VAR_INST
	r_Soc							: REAL;
	fb_SOCLowLimit					: fbValueOutOfRange;
	fb_SOCHighLimit					: fbValueOutOfRange;
	r_SoCMinActual 					: REAL;
	r_SoCMaxActual					: REAL;
	r_deltaSoC						: REAL;
	r_ratio							: REAL;
	r_offset						: REAL;
	
	RS_chargingAllowed				: RS;
	RS_DischargingAllowed			: RS;
END_VAR
//Calculations
r_deltaSoC:= st_params.r_SoCAbsoluteMax - st_params.r_SoCAbsoluteMin;
r_ratio := 1 / SEL(r_deltaSoC=0,r_deltaSoC/100,1);
r_offset := st_params.r_SoCAbsoluteMin * r_Ratio;


//user soc setpoint, first limit user value with 100% and scale to original battery soc 
r_SoCMinActual := (LIMIT(0, set.r_SocMin, set.r_SocMax) + r_Offset) / r_ratio;
r_SoCMaxActual := sel(AutoSOCCalibrationRequired,(LIMIT(set.r_SocMin,set.r_SocMax,100) + r_Offset) / r_ratio, 100);

//Set limit with error when hard limits exceed absolute VDL limits
fb_SOCLowLimit(
	r_var		:= r_SocMinActual, 
	r_min		:= st_params.r_SoCAbsoluteMin, 
	r_max		:= st_params.r_SoCAbsoluteMax,
	r_WhenError := st_params.r_SoCAbsoluteMin,
	b_IsError	=> get.events.b_SoCLowLimitOutOfRange);

fb_SOCHighLimit(
	r_var		:= r_SocMaxActual, 
	r_min		:= st_params.r_SoCAbsoluteMin, 
	r_max		:= st_params.r_SoCAbsoluteMax,
	r_WhenError := st_params.r_SoCAbsoluteMin,
	b_IsError	=> get.events.b_SoCHighLimitOutOfRange);


//Set scaled soc to monitoring
get.BatteryInfo.r_SOCScaled := F_RoundReal(LIMIT(0, get.BatteryInfo.r_SOC * r_ratio - r_offset, 100),1); // set limit to avoid exceed 0 or 100%.

//set scaled kwh discharging remaining
get.BatteryInfo.r_RemainingDischargeEnergyNett := r_deltaSoC/ 100 * get.BatteryInfo.r_RemainingDischargeEnergy;
get.BatteryInfo.r_RemainingChargeEnergyNett := r_deltaSoC/ 100 * get.BatteryInfo.r_RemainingChargeEnergy;

r_Soc := get.BatteryInfo.r_SoC;
//Set Charge only when soft high limit reached
rs_dischargingAllowed(
	set:=r_SoC > (r_SoCMinActual + st_params.r_SocHysteresis),
	Reset1 := r_SoC <= r_SoCMinActual OR get.BatteryInfo.e_BMS_Status = eBMS_Status.FullDischarge,
	Q1 => get.BatteryInfo.b_dischargingAllowed);

//Set discharge only when soft high limit reached
rs_chargingAllowed(
	SET:= r_SoC < (r_SoCMaxActual - st_params.r_SocHysteresis),
	RESET1:= r_SoC >= r_SoCMaxActual OR get.BatteryInfo.e_BMS_Status = eBMS_Status.FullCharge,
	Q1=> get.BatteryInfo.b_chargingAllowed);
END_METHOD

METHOD PRIVATE CalculateTimeRemaining : BOOL
VAR_INPUT
END_VAR

VAR_OUTPUT
END_VAR

VAR_INST
	a_PowerArray			: ARRAY [1..20] OF REAL;
	st_Params_MA			: ST_CTRL_MOVING_AVERAGE_PARAMS;
	ui_filterSize			: UINT := 10;
	fb_SmoothPower			: FB_CTRL_MOVING_AVERAGE;
	r_PowerMA				: REAL;
	r_HoursRemaining		: REAL;
END_VAR
//SMOOTH SETPOINT VALUE SINCE VALUE IS SWITCHED RAPIDLY BETWEEN UPPER AND LOWER GRID LIMIT.
st_Params_MA.tCtrlCycleTime := T#100MS;
	st_Params_MA.tTaskCycleTime := T#1MS;
	st_Params_MA.nWorkArray_SIZEOF := SIZEOF(a_PowerArray);
	st_Params_MA.pWorkArray_ADR	:= ADR(a_PowerArray);
	st_Params_MA.nSamplesToFilter:= ui_filterSize;

fb_SmoothPower(fin:= get.BatteryInfo.r_SystemPower,
				eMode := E_CTRL_MODE.eCTRL_MODE_ACTIVE,
				fout=> r_PowerMA,
				stParams := st_Params_MA);
				
r_HoursRemaining := get.BatteryInfo.r_RemainingDischargeEnergyNett / MAX(1, r_PowerMA);
END_METHOD

METHOD PRIVATE ClearBMSFaults : BOOL
VAR_IN_OUT CONSTANT
	st_params			: ST_BMS_params;
END_VAR

VAR_INST
	WriteRegSet		:	FB_MBWriteSingleReg;
	WriteRegClear	:	FB_MBWriteSingleReg;
	
	bCommBusy	:	BOOL;
	bComError	:	BOOL;
	errID		:	UDINT;
	b_ClearDone	:	BOOL := FALSE;

	w_ClearFault	:	WORD;
	TX1Done 	: 	f_trig;
	
	bCommBusy2	:	BOOL;
	bComError2	:	BOOL;
	errID2		:	UDINT;
	TX2Done 	: 	f_trig;

	ComRetryCounter	:	USINT := 0;	
	
	ResetDelayTimer	: Tp := (PT:=T#500MS);
END_VAR
//Catl says we need to write 1 to clear, then write back to 0 to be able to log new errors.
//This method is called continuously when bms is active. It will usually write zero's.
//If set.b_ClearFault is 1, that will be written. The value will be cleared by this method after the write so next write will be a 0 again.
//With this, a reset cycle takes half a second with the current ComTimer.

ClearBMSFaults := FALSE;

ComTimer(in := NOT(ComTimer.Q OR bCommBusy));

//first write clearing register to 1
WriteRegSet(
	sIPAddr := st_params.IP_BMS,
	nTCPPort := 502,
	nUnitID := 255,//16#FF;
	nMBAddr := 908,
	nValue := 1,
	tTimeOut := t_TimeOut,
	bExecute := ComTimer.Q,
	bBusy => bCommBusy,
	bError => bComError,
	nErrId => errID,
);

TX1Done(CLK := bCommBusy);
b_ClearDone	:= 	TX1Done.Q AND NOT bComError;
ResetDelayTimer(in:=b_ClearDone);
//reset value back to 0 afterwards. CATL requirement
WriteRegClear(
	sIPAddr := st_params.IP_BMS,
	nTCPPort := 502,
	nUnitID := 255,//16#FF;
	nMBAddr := 908,
	nValue := 0,
	tTimeout := T#100MS,
	bExecute := NOT ResetDelayTimer.Q,
	bBusy => bCommBusy2,
	bError => bComError2,
	nErrId => errID2
);

TX2Done(CLK := bCommBusy2);

IF (TX1Done.Q AND bComError) OR (TX2Done.Q AND bComError2) THEN
	ComRetryCounter := ComRetryCounter + 1;
	IF COMRetryCounter > 5 THEN
		b_MBComErrorActive := TRUE;
		ClearBMSFaults := TRUE;
	END_IF
END_IF

IF (TX1Done.Q AND NOT bComError) THEN
	arDatalogEMS[4] := 1;	
END_IF

IF TX2Done.Q AND NOT bComError2 THEN
	arDatalogEMS[4] := 0;	
	b_MBComErrorActive := FALSE;
	ComRetryCounter := 0;
	ClearBMSFaults := TRUE;
END_IF
END_METHOD

METHOD EMSTOP : BOOL
EMSTOP := FALSE;

FBState := ePOUState.EMSTOP;

IF get.MBMU.BatteryStatus.e_BMS_PowerOnStatus <> ePowerOnStatus.On THEN
	EMSTOP := TRUE;
END_IF
END_METHOD

METHOD PRIVATE GetBatteryInfo : BOOL

VAR_IN_OUT
	IN : ST_MBMU_BatterySummary;
	OUT: ST_BMS_BatterySummary;
END_VAR


VAR_INST
	ton_syncPulse : TON := (PT := T#100MS);
	t_SyncTimer	: TIME := T#100MS;
	tof_Release : TOF := (PT:= T#2S);
END_VAR
tof_Release(IN:= get.Events.b_COMMUNICATION_ERROR OR get.MBMU.BatteryStatus.r_SOC > 101);

//set batterysummery data if MBMU gives no shit.
IF ton_syncPulse.Q THEN
	IF NOT tof_Release.Q THEN
		//copy inherited data from original location.
 		MEMCPY(ADR(OUT), ADR(IN), SIZEOF(IN));
		//generate additional data
		CalculateSoCUser(get := get, set := set, st_params:=st_params);
		CalculatedRatings(numberOfStrings:= settings.Configuration.by_NoBatteryStrings);
		CalculateCumulativeValues(get := OUT, t_cycleTime := t_syncTimer);
	ELSE
		out.ar_CellTemperature[0] := -273;
		out.ar_CellTemperature[1] := -273;
		out.ar_CellTemperature[2] := -273;
	END_IF
END_IF
 

ton_syncPulse(IN := NOT ton_syncPulse.Q, PT := t_SyncTimer);
END_METHOD

METHOD PRIVATE GetCellData : BOOL
VAR_IN_OUT CONSTANT
	st_params			: ST_BMS_params;
END_VAR

VAR_INPUT
	SBMUID	:	BYTE;	//SBMU 1-#ofstrings
	CSCID	:	BYTE;	//CSC 1-4
END_VAR

VAR_OUTPUT
	CellVoltages		:	ARRAY[1..52] OF REAL;
	Celltemperatures	:	ARRAY[1..16] OF INT;
	BalanceStatus		:	ARRAY[1..4] OF WORD; //bit per cell?
END_VAR

VAR_INST
	MBReadCellVoltages	: 	FB_MBReadRegs;
	MBReadTemperatures	: 	FB_MBReadRegs;
	MBReadCellBalance	: 	FB_MBReadRegs;
	
//	CellVoltageData		: 	ARRAY[1..52] OF WORD;
	TemperatureData		: 	ARRAY[1..16] OF BYTE;
//	CellBalanceData		: 	ARRAY[1..4] OF WORD;
	
	bCommBusy			:	ARRAY[1..3] OF BOOL;
	bComError			:	ARRAY[1..3] OF BOOL;
	errID				:	ARRAY[1..3] OF UDINT;
	cbRead				:	ARRAY[1..3] OF UDINT;
	TransmissionDone	: 	ARRAY[1..3] OF f_trig;
	
	DataComplete		:	ARRAY[1..3] OF BOOL;
	
	//ComTimer			:	Ton := (PT := TIME#0S500MS);
END_VAR

VAR
	LoopCounter			:	INT;
END_VAR

GetCellData := FALSE;

IF (SBMUID < 1) OR (SBMUID > get.MBMU.by_NumberOfSubSystems) THEN
	GetCellData := TRUE;
	RETURN;
END_IF
IF (CSCID < 1) OR (CSCID > 4) THEN
	GetCellData := TRUE;
	RETURN;
END_IF

ComTimer(in := NOT(ComTimer.Q OR bCommBusy[1] OR bCommBusy[2] OR bCommBusy[3]));

IF ComTimer.Q THEN
	DataComplete[1] := FALSE;
	DataComplete[2] := FALSE;
	DataComplete[3] := FALSE;
END_IF

MBReadCellVoltages(
sIPAddr := st_params.IP_BMS,
nTCPPort := 502,
nUnitID := 255,//16#FF;
nMBAddr := (SBMUID*1024)+128+(52*(CSCID-1)),	//SBMU 1, module 1, start at 0x0480, increment 52 per module & 1024 per sbmu
nQuantity := 52,
cbLength := SIZEOF(CellVoltages),
pDestAddr := ADR(CellVoltages),
bExecute := ComTimer.Q,
bBusy => bCommBusy[1],
bError => bComError[1],
nErrId => errID[1],
cbRead => cbRead[1],
tTimeOut := t_TimeOut,
);

MBReadTemperatures(
sIPAddr := st_params.IP_BMS,
nTCPPort := 502,
nUnitID := 1,//16#FF;
nMBAddr := (SBMUID*1024)+704+(8*(CSCID-1)),	//SBMU 1, module 1, start at 0x06c0, increment 8 (16 byte) per module & 1024 per sbmu
nQuantity := 8*2,
cbLength := SIZEOF(TemperatureData),
pDestAddr := ADR(TemperatureData),
bExecute := ComTimer.Q,
bBusy => bCommBusy[2],
bError => bComError[2],
nErrId => errID[2],
cbRead => cbRead[2],
tTimeOut := t_TimeOut,
);

MBReadTemperatures(
sIPAddr := st_params.IP_BMS,
nTCPPort := 502,
nUnitID := 1,//16#FF;
nMBAddr := (SBMUID*1024)+912+(4*(CSCID-1)),	//SBMU 1, module 1, start at 0x0790, increment 4 per module & 1024 per sbmu
											//not sure if CSC2 starts at address 4, or immediatly follows after last cell of csc1.
nQuantity := 4*2,
cbLength := SIZEOF(BalanceStatus),
pDestAddr := ADR(BalanceStatus),
bExecute := ComTimer.Q,
bBusy => bCommBusy[3],
bError => bComError[3],
nErrId => errID[3],
cbRead => cbRead[3],
tTimeOut := t_TimeOut,
);

TransmissionDone[1](clk:=bCommBusy[1]);
TransmissionDone[2](clk:=bCommBusy[2]);
TransmissionDone[3](clk:=bCommBusy[3]);

IF TransmissionDone[1].Q AND NOT bComError[1] THEN
	DataComplete[1] := TRUE;
END_IF

IF TransmissionDone[2].Q AND NOT bComError[2] THEN
	FOR loopcounter := 1 TO 16 BY 1 DO
		Celltemperatures[loopcounter] := TemperatureData[loopcounter]-50;
	END_FOR
	DataComplete[2] := TRUE;
END_IF

IF TransmissionDone[1].Q AND NOT bComError[1] THEN
	DataComplete[3] := TRUE;
END_IF

GetCellData := DataComplete[1] AND DataComplete[2] AND DataComplete[3];
END_METHOD

METHOD GetDiagnostics 
VAR_IN_OUT
	AddError		: ARRAY [*] OF FB_AddErrorST;
	a_ActiveEvents	: ARRAY [*] OF ST_ErrorStruct;
	w_Index			: WORD;
END_VAR
(*BMS errors (sunspec)*)
	(*BMS Communication error*)		AddError[w_Index](
			b_ErrorTrig				:= get.Events.b_COMMUNICATION_ERROR,
			out_ST_Error			:= a_ActiveEvents[w_Index],
			w_ErrorID				:= 1,
			e_ObjectID				:= e_id,						//only first call set object ID.
			s_Message				:= 'communication error',
			e_sev					:= eSeverity.QuickShutdown,	//<-- maybe normal shutdown?
			b_AutoClear				:= FALSE,
			t_TriggerTime			:= TIME#10S,
			e_ErrAckAccess			:= eErrAckAccess.Operator
			);
		w_Index := w_Index +1;
		
	(*Configuration fault*)		AddError[w_Index](
			b_ErrorTrig				:= get.Events.b_CONFIGURATION_ALARM,
			out_ST_Error			:= a_ActiveEvents[w_Index],
			w_ErrorID				:= 2,
			s_Message				:= 'configuration error',
			e_sev					:= eSeverity.NormalShutdown,
			b_AutoClear				:= FALSE,
			e_ErrAckAccess			:= eErrAckAccess.VDL
			//in_t_TriggerTime		:= TIME#500MS,
			//in_e_ErrAckAccess		:= TRUE,
			);
		w_Index := w_Index +1;
	
	(*Configuration warning*)		AddError[w_Index](
			b_ErrorTrig				:= get.Events.b_CONFIGURATION_WARNING,
			out_ST_Error			:= a_ActiveEvents[w_Index],
			w_ErrorID				:= 3,
			s_Message				:= 'configuration error',
			e_sev					:= eSeverity.Warning,
			b_AutoClear				:= FALSE,
			e_ErrAckAccess			:= eErrAckAccess.Operator
			//in_t_TriggerTime		:= TIME#500MS,
			//in_e_ErrAckAccess		:= TRUE,
			);
		w_Index := w_Index +1;
		
	(*Contactor fault*)		AddError[w_Index](
			b_ErrorTrig				:= get.Events.b_CONTACTOR_ERROR,
			out_ST_Error			:= a_ActiveEvents[w_Index],
			w_ErrorID				:= 4,
			s_Message				:= 'contactor fault',
			e_sev					:= eSeverity.QuickShutdown,
			b_AutoClear				:= FALSE,
			e_ErrAckAccess			:= eErrAckAccess.Operator
			//in_t_TriggerTime		:= TIME#500MS,
			//in_e_ErrAckAccess		:= TRUE,
			);
		w_Index := w_Index +1;
		
	(*Current imbalance warning*)		AddError[w_Index](						//unused, will always be false
			b_ErrorTrig				:= get.Events.b_CURRENT_IMBALANCE_WARNING,
			out_ST_Error			:= a_ActiveEvents[w_Index],
			w_ErrorID				:= 5,
			s_Message				:= 'current imbalance warning',
			e_sev					:= eSeverity.Warning,
			b_AutoClear				:= FALSE,
			e_ErrAckAccess			:= eErrAckAccess.General
			//in_t_TriggerTime		:= TIME#500MS,
			);
		w_Index := w_Index +1;
		
	(*Fan error*)		AddError[w_Index](
			b_ErrorTrig				:= get.Events.b_FAN_ERROR,
			out_ST_Error			:= a_ActiveEvents[w_Index],
			w_ErrorID				:= 6,
			s_Message				:= 'fan error',
			e_sev					:= eSeverity.NormalShutdown,
			b_AutoClear				:= FALSE,
			//in_t_TriggerTime		:= TIME#500MS,
			e_ErrAckAccess			:= eErrackAccess.Operator
			);
		w_Index := w_Index +1;

	(*Ground fault*)		AddError[w_Index](
			b_ErrorTrig			:= get.Events.b_GROUND_FAULT,		//unused, will always be false
			out_ST_Error			:= a_ActiveEvents[w_Index],
			w_ErrorID					:= 7,
			s_Message				:= 'insulation fault',
			e_sev					:= eSeverity.Quickshutdown,
			b_AutoClear				:= FALSE,
			//in_t_TriggerTime		:= TIME#500MS,
			//in_e_ErrAckAccess		:= TRUE,
			);
		w_Index := w_Index +1;

	(*Door open error*)		AddError[w_Index](							//unused, will always be false
			b_ErrorTrig			:= get.Events.b_OPEN_DOOR_ERROR,
			out_ST_Error			:= a_ActiveEvents[w_Index],
			w_ErrorID					:= 8,
			s_Message				:= 'door open',
			e_sev					:= eSeverity.NormalShutdown,
			b_AutoClear				:= TRUE,
			//in_t_TriggerTime		:= TIME#500MS,
			//in_e_ErrAckAccess		:= TRUE,
			);
		w_Index := w_Index +1;

	(*misc alarm*)		AddError[w_Index](							
			b_ErrorTrig			:= get.Events.b_OTHER_ALARM,
			out_ST_Error			:= a_ActiveEvents[w_Index],
			w_ErrorID					:= 9,
			s_Message				:= 'miscellaneous error',
			e_sev					:= eSeverity.NormalShutdown,
			b_AutoClear				:= FALSE,
			//in_t_TriggerTime		:= TIME#500MS,
			//in_e_ErrAckAccess		:= TRUE,
			);
		w_Index := w_Index +1;
		
	(*misc warning*)		AddError[w_Index](							
			b_ErrorTrig			:= get.Events.b_OTHER_WARNING,
			out_ST_Error			:= a_ActiveEvents[w_Index],
			w_ErrorID					:= 10,
			s_Message				:= 'miscellaneous warning',
			e_sev					:= eSeverity.Warning,
			b_AutoClear				:= TRUE,
			//in_t_TriggerTime		:= TIME#500MS,
			//in_e_ErrAckAccess		:= TRUE,
			);
		w_Index := w_Index +1;

	(*Overcharge current alarm*)		AddError[w_Index](							
			b_ErrorTrig			:= get.Events.b_OVER_CHARGE_CURRENT_ALARM,
			out_ST_Error			:= a_ActiveEvents[w_Index],
			w_ErrorID					:= 11,
			s_Message				:= 'charge current too high error',
			e_sev					:= eSeverity.NormalShutdown,			
			b_AutoClear				:= FALSE,									
			//in_t_TriggerTime		:= TIME#500MS,
			//in_e_ErrAckAccess		:= TRUE,
			);
		w_Index := w_Index +1;
		
	(*Overcharge current warning*)		AddError[w_Index](							
			b_ErrorTrig			:= get.Events.b_OVER_CHARGE_CURRENT_WARNING,
			out_ST_Error			:= a_ActiveEvents[w_Index],
			w_ErrorID					:= 12,
			s_Message				:= 'charge current high warning',
			e_sev					:= eSeverity.Warning,				//<-- Powerstack should lower the power
			b_AutoClear				:= TRUE,								
			//in_t_TriggerTime		:= TIME#500MS,
			//in_e_ErrAckAccess		:= TRUE,
			);
		w_Index := w_Index +1;
		
	(*OverDischarge current Alarm*)		AddError[w_Index](							
			b_ErrorTrig			:= get.Events.b_OVER_DISCHARGE_CURRENT_ALARM,
			out_ST_Error			:= a_ActiveEvents[w_Index],
			w_ErrorID					:= 13,
			s_Message				:= 'discharge current too high error',
			e_sev					:= eSeverity.NormalShutdown,				
			b_AutoClear				:= FALSE,								
			//in_t_TriggerTime		:= TIME#500MS,
			//in_e_ErrAckAccess		:= TRUE,
			);

		w_Index := w_Index +1;
		
	(*OverDischarge current warning*)		AddError[w_Index](							
			b_ErrorTrig			:= get.Events.b_OVER_DISCHARGE_CURRENT_WARNING,
			out_ST_Error			:= a_ActiveEvents[w_Index],
			w_ErrorID					:= 14,
			s_Message				:= 'discharge current high warning',
			e_sev					:= eSeverity.Warning,				//<-- Powerstack should lower the power
			b_AutoClear				:= TRUE,								
			//in_t_TriggerTime		:= TIME#500MS,
			//in_e_ErrAckAccess		:= TRUE,
			);
		w_Index := w_Index +1;
		
	(*Overcharge r_SOC error*)		AddError[w_Index](							//unused, will remain false
			b_ErrorTrig			:= get.Events.b_OVER_SOC_MAX_ALARM AND NOT st_params.b_DisableSOCAlarm,
			out_ST_Error			:= a_ActiveEvents[w_Index],
			w_ErrorID					:= 15,
			s_Message				:= 'SOC too high error',
			e_sev					:= eSeverity.NormalShutdown,				
			b_AutoClear			:= FALSE,								
			//in_t_TriggerTime		:= TIME#500MS,
			//in_e_ErrAckAccess		:= TRUE,
			);
		w_Index := w_Index +1;
		
	(*Overcharge r_SOC error*)		AddError[w_Index](							//unused, will remain false
			b_ErrorTrig			:= get.Events.b_OVER_SOC_MAX_WARNING,
			out_ST_Error			:= a_ActiveEvents[w_Index],
			w_ErrorID					:= 16,
			s_Message				:= 'SOC high warning',
			e_sev					:= eSeverity.Warning,				
			b_AutoClear				:= TRUE,								
			//in_t_TriggerTime		:= TIME#500MS,
			//in_e_ErrAckAccess		:= TRUE,
			);
		w_Index := w_Index +1;
		
	(*OverDischarge r_SOC error*)		AddError[w_Index](							
			b_ErrorTrig			:= get.Events.b_UNDER_SOC_MIN_ALARM AND NOT st_params.b_DisableSOCAlarm,
			out_ST_Error			:= a_ActiveEvents[w_Index],
			w_ErrorID					:= 17,
			s_Message				:= 'SOC too low error',
			e_sev					:= eSeverity.NormalShutdown,				
			b_AutoClear			:= FALSE,								
			//in_t_TriggerTime		:= TIME#500MS,
			//in_e_ErrAckAccess		:= TRUE,
			);
		w_Index := w_Index +1;
		
	(*OverDischarge r_SOC error*)		AddError[w_Index](							
			b_ErrorTrig			:= get.Events.b_UNDER_SOC_MIN_WARNING,
			out_ST_Error			:= a_ActiveEvents[w_Index],
			w_ErrorID					:= 18,
			s_Message				:= 'SOC low warning',
			e_sev					:= eSeverity.Warning,				
			b_AutoClear				:= TRUE,								
			//in_t_TriggerTime		:= TIME#500MS,
			//in_e_ErrAckAccess		:= TRUE,
			);
		w_Index := w_Index +1;
		
	(*OverTemperature error*)		AddError[w_Index](							
			b_ErrorTrig			:= get.Events.b_OVER_TEMP_ALARM,
			out_ST_Error			:= a_ActiveEvents[w_Index],
			w_ErrorID					:= 19,
			s_Message				:= 'overtemperature alarm',
			e_sev					:= eSeverity.NormalShutdown,				
			b_AutoClear			:= FALSE,
			b_SMSEnableVDL		:= TRUE,								
			//in_t_TriggerTime		:= TIME#500MS,
			//in_e_ErrAckAccess		:= TRUE,
			);
		w_Index := w_Index +1;		

	(*OverTemperature warning*)		AddError[w_Index](							
			b_ErrorTrig			:= get.Events.b_OVER_TEMP_WARNING,
			out_ST_Error			:= a_ActiveEvents[w_Index],
			w_ErrorID					:= 20,
			s_Message				:= 'overtemperature warning',
			e_sev					:= eSeverity.Warning,				
			b_AutoClear			:= FALSE,								
			//in_t_TriggerTime		:= TIME#500MS,
			//in_e_ErrAckAccess		:= TRUE,
			);
		w_Index := w_Index +1;
	
	(*OverVoltage error*)		AddError[w_Index](							
			b_ErrorTrig			:= get.Events.b_OVER_VOLT_ALARM,
			out_ST_Error			:= a_ActiveEvents[w_Index],
			w_ErrorID					:= 21,
			s_Message				:= 'overvoltage error',
			e_sev					:= eSeverity.NormalShutdown,
			b_SMSEnableVDL		:= TRUE,				
			b_AutoClear			:= FALSE,								
			//in_t_TriggerTime		:= TIME#500MS,
			//in_e_ErrAckAccess		:= TRUE,
			);
		w_Index := w_Index +1;		

	(*OverVoltage warning*)		AddError[w_Index](							
			b_ErrorTrig			:= get.Events.b_OVER_VOLT_WARNING,
			out_ST_Error			:= a_ActiveEvents[w_Index],
			w_ErrorID					:= 22,
			s_Message				:= 'overvoltage warning',
			e_sev					:= eSeverity.Warning,				
			b_AutoClear			:= FALSE,								
			//in_t_TriggerTime		:= TIME#500MS,
			//in_e_ErrAckAccess		:= TRUE,
			);
		w_Index := w_Index +1;
		
	(*Temperature imbalance error*)		AddError[w_Index](							
			b_ErrorTrig			:= get.Events.b_TEMPERATURE_IMBALANCE_ALARM,
			out_ST_Error			:= a_ActiveEvents[w_Index],
			w_ErrorID					:= 23,
			s_Message				:= 'temperature imbalance error',
			e_sev					:= eSeverity.NormalShutdown,				
			b_AutoClear			:= FALSE,								
			//in_t_TriggerTime		:= TIME#500MS,
			//in_e_ErrAckAccess		:= TRUE,
			);
		w_Index := w_Index +1;		

	(*Temperature imbalance warning*)		AddError[w_Index](							
			b_ErrorTrig			:= get.Events.b_TEMPERATURE_IMBALANCE_WARNING,
			out_ST_Error			:= a_ActiveEvents[w_Index],
			w_ErrorID					:= 24,
			s_Message				:= 'temperature imbalance warning',
			e_sev					:= eSeverity.Warning,				
			b_AutoClear			:= FALSE,								
			//in_t_TriggerTime		:= TIME#500MS,
			//in_e_ErrAckAccess		:= TRUE,
			);
		w_Index := w_Index +1;

	(*Under Temperature error*)		AddError[w_Index](							
			b_ErrorTrig			:= get.Events.b_UNDER_TEMP_ALARM,
			out_ST_Error			:= a_ActiveEvents[w_Index],
			w_ErrorID					:= 25,
			s_Message				:= 'temperature low error',
			e_sev					:= eSeverity.NormalShutdown,				
			b_AutoClear			:= FALSE,								
			//in_t_TriggerTime		:= TIME#500MS,
			//in_e_ErrAckAccess		:= TRUE,
			);
		w_Index := w_Index +1;		

	(*Under Temperature warning*)		AddError[w_Index](							
			b_ErrorTrig			:= get.Events.b_UNDER_TEMP_WARNING,
			out_ST_Error			:= a_ActiveEvents[w_Index],
			w_ErrorID					:= 26,
			s_Message				:= 'temperature low warning',
			e_sev					:= eSeverity.Warning,				
			b_AutoClear			:= TRUE,								
			//in_t_TriggerTime		:= TIME#500MS,
			//in_e_ErrAckAccess		:= TRUE,
			);
		w_Index := w_Index +1;

	(*Under Temperature error*)		AddError[w_Index](							
			b_ErrorTrig			:= get.Events.b_UNDER_VOLT_ALARM,
			out_ST_Error			:= a_ActiveEvents[w_Index],
			w_ErrorID					:= 27,
			s_Message				:= 'undervoltage error',
			e_sev					:= eSeverity.NormalShutdown,				
			b_AutoClear			:= FALSE,								
			//in_t_TriggerTime		:= TIME#500MS,
			//in_e_ErrAckAccess		:= TRUE,
			);
		w_Index := w_Index +1;		

	(*Under Temperature warning*)		AddError[w_Index](							
			b_ErrorTrig			:= get.Events.b_UNDER_VOLT_WARNING,
			out_ST_Error			:= a_ActiveEvents[w_Index],
			w_ErrorID					:= 28,
			s_Message				:= 'undervoltage warning',
			e_sev					:= eSeverity.Warning,				
			b_AutoClear			:= FALSE,								
			//in_t_TriggerTime		:= TIME#500MS,
			//in_e_ErrAckAccess		:= TRUE,
			);
		w_Index := w_Index +1;
		
	(*Battery voltage imbalance warning*)		AddError[w_Index](							
			b_ErrorTrig			:= get.Events.b_VOLTAGE_IMBALANCE_WARNING,
			out_ST_Error			:= a_ActiveEvents[w_Index],
			w_ErrorID					:= 29,
			s_Message				:= 'voltage imbalance warning',
			e_sev					:= eSeverity.Warning,				
			b_AutoClear			:= FALSE,								
			//in_t_TriggerTime		:= TIME#500MS,
			);
		w_Index := w_Index +1;	
		
		(*Battery voltage imbalance warning*)		AddError[w_Index](							
			b_ErrorTrig			:= get.Events.b_SocHighLimitOutOfRange,
			out_ST_Error			:= a_ActiveEvents[w_Index],
			w_ErrorID					:= 30,
			s_Message				:= 'SOC upper limit out of range',
			e_sev					:= eSeverity.info,				
			b_AutoClear			:= TRUE,								
			);
		w_Index := w_Index +1;	
		
				(*Battery voltage imbalance warning*)		AddError[w_Index](							
			b_ErrorTrig			:= get.Events.b_SocLowLimitOutOfRange,
			out_ST_Error			:= a_ActiveEvents[w_Index],
			w_ErrorID					:= 31,
			s_Message				:= 'SOC lower limit out of range',
			e_sev					:= eSeverity.info,				
			b_AutoClear			:= TRUE,								
			);
		w_Index := w_Index +1;	
	
(*Battery PRECHARGE FAULT*)		AddError[w_Index](							
			b_ErrorTrig			:= get.Events.b_POWERONFAULT,
			out_ST_Error			:= a_ActiveEvents[w_Index],
			w_ErrorID					:= 32,
			s_Message				:= 'precharge fault',
			e_sev					:= eSeverity.warning,				
			b_AutoClear			:= TRUE,								
			);
		w_Index := w_Index +1;	
		
(*Battery power off fault*)		AddError[w_Index](							
			b_ErrorTrig			:= get.Events.b_POWEROFFFAULT,
			out_ST_Error			:= a_ActiveEvents[w_Index],
			w_ErrorID					:= 33,
			s_Message				:= 'poweroff fault',
			e_sev					:= eSeverity.Quickshutdown,				
			b_AutoClear			:= FALSE,								
			);
		w_Index := w_Index +1;	
		
(*Disconnector Off*)		AddError[w_Index](							
			b_ErrorTrig			:= get.Events.b_DISCONNECTOR_OFF,
			out_ST_Error			:= a_ActiveEvents[w_Index],
			w_ErrorID					:= 35,
			s_Message				:= 'HV disconnector(s) off position',
			e_sev					:= eSeverity.Normalshutdown,				
			b_AutoClear			:= FALSE,								
			);
		w_Index := w_Index +1;
		
(*SBMU1 com failed*)		AddError[w_Index](							
			b_ErrorTrig				:= get.Events.b_SBMUCommError[0],
			out_ST_Error			:= a_ActiveEvents[w_Index],
			w_ErrorID				:= 36,
			s_Message				:= 'SBMU 1 Com Warning',
			e_sev					:= eSeverity.Warning,				
			b_AutoClear				:= TRUE,
			t_TriggerTime			:= TIME#5S,								
			);
		w_Index := w_Index +1;

(*SBMU2 com failed*)		AddError[w_Index](							
			b_ErrorTrig				:= get.Events.b_SBMUCommError[1],
			out_ST_Error			:= a_ActiveEvents[w_Index],
			w_ErrorID				:= 37,
			s_Message				:= 'SBMU 2 Com Warning',
			e_sev					:= eSeverity.Warning,				
			b_AutoClear				:= TRUE,
			t_TriggerTime			:= TIME#5S,								
			);
		w_Index := w_Index +1;

(*SBMU3 com failed*)		AddError[w_Index](							
			b_ErrorTrig				:= get.Events.b_SBMUCommError[2],
			out_ST_Error			:= a_ActiveEvents[w_Index],
			w_ErrorID				:= 38,
			s_Message				:= 'SBMU 3 Com Warning',
			e_sev					:= eSeverity.Warning,				
			b_AutoClear				:= TRUE,
			t_TriggerTime			:= TIME#5S,								
			);
		w_Index := w_Index +1;

(*SBMU4 com failed*)		AddError[w_Index](							
			b_ErrorTrig				:= get.Events.b_SBMUCommError[3],
			out_ST_Error			:= a_ActiveEvents[w_Index],
			w_ErrorID				:= 39,
			s_Message				:= 'SBMU 4 Com Warning',
			e_sev					:= eSeverity.Warning,				
			b_AutoClear				:= TRUE,
			t_TriggerTime			:= TIME#5S,								
			);
		w_Index := w_Index +1;
		
(*SBMU1 failed to connect HV*)		AddError[w_Index](							
			b_ErrorTrig				:= get.Events.b_SBMUFailedToConnect[0],
			out_ST_Error			:= a_ActiveEvents[w_Index],
			w_ErrorID				:= 40,
			s_Message				:= 'SBMU 1 failed to connect to DC bus',
			e_sev					:= eSeverity.Warning,				
			b_AutoClear				:= TRUE,
			t_TriggerTime			:= TIME#5S,								
			);
		w_Index := w_Index +1;

(*SBMU2 com failed*)		AddError[w_Index](							
			b_ErrorTrig				:= get.Events.b_SBMUFailedToConnect[1],
			out_ST_Error			:= a_ActiveEvents[w_Index],
			w_ErrorID				:= 41,
			s_Message				:= 'SBMU 2 failed to connect to DC bus',
			e_sev					:= eSeverity.Warning,				
			b_AutoClear				:= TRUE,
			t_TriggerTime			:= TIME#5S,								
			);
		w_Index := w_Index +1;

(*SBMU3 com failed*)		AddError[w_Index](							
			b_ErrorTrig				:= get.Events.b_SBMUFailedToConnect[2],
			out_ST_Error			:= a_ActiveEvents[w_Index],
			w_ErrorID				:= 42,
			s_Message				:= 'SBMU 3 failed to connect to DC bus',
			e_sev					:= eSeverity.Warning,				
			b_AutoClear				:= TRUE,
			t_TriggerTime			:= TIME#5S,								
			);
		w_Index := w_Index +1;

(*SBMU4 com failed*)		AddError[w_Index](							
			b_ErrorTrig				:= get.Events.b_SBMUFailedToConnect[3],
			out_ST_Error			:= a_ActiveEvents[w_Index],
			w_ErrorID				:= 43,
			s_Message				:= 'SBMU 4 failed to connect to DC bus',
			e_sev					:= eSeverity.Warning,				
			b_AutoClear				:= TRUE,
			t_TriggerTime			:= TIME#5S,								
			);
		w_Index := w_Index +1;
		
		
(*SOC too low for conditioning*)		AddError[w_Index](							
			b_ErrorTrig				:= NOT b_InternalHVDCAllowed,
			out_ST_Error			:= a_ActiveEvents[w_Index],
			w_ErrorID				:= 44,
			s_Message				:= 'SOC low warning. Internal Conditioning disabled',
			e_sev					:= eSeverity.Warning,				
			b_AutoClear				:= TRUE,
			t_TriggerTime			:= TIME#5S,								
			);
		w_Index := w_Index +1;
END_METHOD

METHOD PRIVATE GetMBMUData : BOOL
VAR_IN_OUT CONSTANT
	st_params			: ST_BMS_params;
END_VAR


VAR_INST
	
	MBReadMBMU			: 	FB_MBReadRegs;
	MBMUData 			: 	ARRAY[0..52] OF WORD;
	bCommBusy			:	BOOL;
	bComError			:	BOOL;
	errID				:	UDINT;
	cbRead				:	UDINT;
	TransmissionDone	: 	f_trig;
	COMretryCounter		:	USINT := 0;
	//ComTimer			:	Ton := (PT := TIME#100MS);
END_VAR

VAR
	Counter				:	INT;
END_VAR
//read mbmu data every 100ms

GetMBMUData := FALSE;

ComTimer(in := NOT(ComTimer.Q OR bCommBusy));

MBReadMBMU(
sIPAddr := st_params.IP_BMS,
nTCPPort := 502,
nUnitID := 255,//16#FF;
nMBAddr := 0,
nQuantity := 53,
cbLength := SIZEOF(MBMUData),
pDestAddr := ADR(MBMUData),
bExecute := ComTimer.Q,
bBusy => bCommBusy,
bError => bComError,
nErrId => errID,
cbRead => cbRead,
tTimeout := t_TimeOut,
);

TransmissionDone(CLK := bCommBusy);

IF TransmissionDone.Q THEN
	IF NOT bComError THEN
		MEMCPY(ADR(get.MBMU.GeneralSBMUStatus[0]), ADR(MBMUData[0]), 32);	//0x0000 - 0x000f
		MEMCPY(ADR(get.MBMU.MBMUStatus[0]), ADR(MBMUData[16]), 32);			//0x0010 - 0x001f
	
		get.MBMU.BatteryStatus.r_SystemVoltage := WORD_TO_REAL(MBMUData[32])/10; 						//0-1500V with 0.1V/bit
		get.MBMU.BatteryStatus.r_SystemCurrent := WORD_TO_REAL(MBMUData[33])-20000; 					//-20k .. +20k kW in 1kW/bit steps
		
		get.MBMU.BatteryStatus.r_SOC := WORD_TO_REAL(MBMUData[34])/10; 								//0-100% with 0.1%/bit;
		get.MBMU.BatteryStatus.r_SOH := WORD_TO_REAL(MBMUData[35])/10; 								//0-100% with 0.1%/bit;
		
		get.MBMU.BatteryStatus.ar_CellVoltage[eSubValues.Maximum] := WORD_TO_REAL(MBMUData[36])/1000;	//0-5v with 0.001v/bit;
		get.MBMU.BatteryStatus.ar_CellVoltage[eSubValues.Minimum] := WORD_TO_REAL(MBMUData[37])/1000;	//0-5v with 0.001v/bit;
		get.MBMU.BatteryStatus.ar_CellVoltage[eSubValues.Average] := WORD_TO_REAL(MBMUData[38])/1000;	//0-5v with 0.001v/bit;
		
		get.MBMU.BatteryStatus.ar_CellTemperature[eSubValues.Maximum] := WORD_TO_REAL(MBMUData[39])-50;	//-50..200gr with 1gr/bit;
		get.MBMU.BatteryStatus.ar_CellTemperature[eSubValues.Minimum] := WORD_TO_REAL(MBMUData[40])-50;	//-50..200gr with 1gr/bit;
		get.MBMU.BatteryStatus.ar_CellTemperature[eSubValues.Average] := WORD_TO_REAL(MBMUData[41])-50;	//-50..200gr with 1gr/bit;
		
		get.MBMU.BatteryStatus.r_MaxChargeCurrentAllowed := WORD_TO_REAL(MBMUData[42])-20000;			//-20k .. +20k A in 1A/bit steps
		get.MBMU.BatteryStatus.r_MaxDischargeCurrentAllowed := WORD_TO_REAL(MBMUData[43])-20000;			//-20k .. +20k A in 1A/bit steps
		
		get.MBMU.BatteryStatus.r_MaxChargePowerAllowed := WORD_TO_REAL(MBMUData[44])-20000;				//-20k .. +20k kW in 1kW/bit steps
		get.MBMU.BatteryStatus.r_MaxDischargePowerAllowed := WORD_TO_REAL(MBMUData[45])-20000;			//-20k .. +20k kW in 1kW/bit steps
		
		get.MBMU.BatteryStatus.r_SystemPower	:= 	WORD_TO_REAL(MBMUData[46])-20000;						//-20k .. +20k kW in 1kW/bit steps
		get.MBMU.BatteryStatus.r_ChargeSOE	:=	WORD_TO_REAL(MBMUData[47])/10;
		get.MBMU.BatteryStatus.r_DischargeSOE	:=	WORD_TO_REAL(MBMUData[48])/10;
		
		get.MBMU.BatteryStatus.r_RemainingChargeEnergy	:=	WORD_TO_REAL(MBMUData[49]) *2;
		get.MBMU.BatteryStatus.r_RemainingDischargeEnergy	:=	WORD_TO_REAL(MBMUData[50]) *2;
		
		get.MBMU.BatteryStatus.r_MaxSystemVoltageAllowed := WORD_TO_REAL(MBMUData[51])/10; 			//0-1500V with 0.1V/bit
		get.MBMU.BatteryStatus.r_MinSystemVoltageAllowed := WORD_TO_REAL(MBMUData[52])/10; 			//0-1500V with 0.1V/bit
			
		memcpy(ADR(arDatalogMBMU), ADR(MBMUData), 92);	//0-46
		
		GetMBMUData := TRUE;
		COMretryCounter := 0;
		b_MBComErrorActive := FALSE;
	ELSE
		COMretryCounter := COMretryCounter +1;
		IF COMRetryCounter > 5 THEN
			b_MBComErrorActive := TRUE;
		END_IF
	END_IF
END_IF
END_METHOD

METHOD PRIVATE GetMBMUStaticSystemData : BOOL
VAR_IN_OUT CONSTANT
	st_params			: ST_BMS_params;
END_VAR

VAR_INST
	MBReadBMS			: 	FB_MBReadRegs;
	DataBuffer 			: 	ARRAY[0..31] OF WORD;
	
	bCommBusy			:	BOOL;
	bComError			:	BOOL;
	errID				:	UDINT;
	cbRead				:	UDINT;
	
	TransmissionDone 	: 	f_trig;
	COMretryCounter		:	USINT := 0;
	//ComTimer			:	Ton := (PT := TIME#200ms);
END_VAR

//Read ETH+MBMU SW/HW version at init.
GetMBMUStaticSystemData := FALSE;

ComTimer(in := NOT(ComTimer.Q));

MBReadBMS(
sIPAddr := st_params.IP_BMS,
nTCPPort := 502,
nUnitID := 255,//16#FF;
nMBAddr := 256,
nQuantity := 32,
cbLength := SIZEOF(DataBuffer),
pDestAddr := ADR(DataBuffer),
bExecute := ComTimer.Q,
tTimeout := t_TimeOut,
bBusy => bCommBusy,
bError => bComError,
nErrId => errID,
cbRead => cbRead
);

TransmissionDone(CLK := bCommBusy);

IF TransmissionDone.Q THEN
	IF NOT bComError THEN
		memcpy(destAddr := ADR(get.MBMU.s_MBMU_SWVer), SrcAddr := ADR(DataBuffer[0]), n := 16);
		memcpy(destAddr  := ADR(get.MBMU.s_MBMU_HWVer), SrcAddr := ADR(DataBuffer[8]), n := 16);
		memcpy(destAddr  := ADR(get.MBMU.s_ETH_SWVer), SrcAddr := ADR(DataBuffer[16]), n := 16);
		memcpy(destAddr  := ADR(get.MBMU.r_ETH_HWVer), SrcAddr :=ADR( DataBuffer[24]), n := 16);
		GetMBMUStaticSystemData := TRUE;
		COMretryCounter := 0;
		b_MBComErrorActive := FALSE;
	ELSE
		COMretryCounter := COMretryCounter +1;
		IF COMRetryCounter > 5 THEN
			b_MBComErrorActive := TRUE;
		END_IF
	END_IF
END_IF
END_METHOD

METHOD PRIVATE GetSBMUData : BOOL
VAR_IN_OUT CONSTANT
	st_params			: ST_BMS_params;
END_VAR

VAR_INST
	MBReadSBMU		: 	FB_MBReadRegs;
	DataBuffer		:	ARRAY[0..91] OF WORD;
	bCommBusy		:	BOOL;
	bComError		:	BOOL;
	errID			:	UDINT;
	cbRead			:	UDINT;
	CommDone		: 	f_trig;
	tempSBMUStatus	:	WORD;
	SBMUCounter		: 	USINT	:=	0;
	//ComTimer			:	Ton := (PT := TIME#100MS);
END_VAR

VAR
	b_MainRelayClosed 		: 	BOOL;
	b_PrechargeRelayClosed	:	BOOL;
	ui_SBMUCounter			:	uint;
END_VAR
GetSBMUData := FALSE;

ComTimer(in := NOT(ComTimer.Q OR bCommbusy));

MBReadSBMU(
	sIPAddr := st_params.IP_BMS,
	nTCPPort := 502,
	nUnitID := 255,//16#FF;
	nMBAddr := 1024*(SBMUcounter+1),
	nQuantity := 91,
	cbLength := SIZEOF(DataBuffer),
	pDestAddr := ADR(DataBuffer),
	bExecute := ComTimer.Q,
	tTimeout := t_TimeOut,
	bBusy => bCommBusy,
	bError => bComError,
	nErrId => errID,
	cbRead => cbRead
);
	
CommDone(CLK := bCommBusy);
	
IF CommDone.Q THEN
	IF NOT bComError THEN
		get.SBMU[SBMUcounter].w_SystemWarning := DataBuffer[0];
		get.SBMU[SBMUcounter].SystemAlarm[0] := DataBuffer[1];
		get.SBMU[SBMUcounter].SystemAlarm[1] := DataBuffer[2];
		get.SBMU[SBMUcounter].SystemAlarm[2] := DataBuffer[3];
		
		get.SBMU[SBMUcounter].b_PrechargeRelayClosed 	:= WORD_TO_BOOL(DataBuffer[16]);
		get.SBMU[SBMUcounter].b_MainPosRelayClosed	 	:= WORD_TO_BOOL(DataBuffer[17]);
		get.SBMU[SBMUcounter].b_MainNegRelayClosed		:= WORD_TO_BOOL(DataBuffer[18]);
		get.SBMU[SBMUcounter].b_ControlBoxFanOn 			:= WORD_TO_BOOL(DataBuffer[19]);
		get.SBMU[SBMUcounter].b_BalanceStatus 			:= WORD_TO_BOOL(DataBuffer[20]);
		
		get.SBMU[SBMUcounter].BatteryStatus.r_SystemVoltage := WORD_TO_REAL(DataBuffer[32])/10;	//0-1500V with 0.1V/bit
		get.SBMU[SBMUcounter].BatteryStatus.r_SystemCurrent := (WORD_TO_REAL(DataBuffer[34])/10)-2000; 	//-2k .. +2k A in 0.1A/bit steps
		
		get.SBMU[SBMUcounter].BatteryStatus.r_SOC := WORD_TO_REAL(DataBuffer[35])/10; 			//0-100% with 0.1%/bit;
		get.SBMU[SBMUcounter].BatteryStatus.r_SOH := WORD_TO_REAL(DataBuffer[36])/10;				//0-100% with 0.1%/bit;
		
		get.SBMU[SBMUcounter].BatteryStatus.ar_CellVoltage[eSubValues.Maximum] := WORD_TO_REAL(DataBuffer[37])/1000;	//0-5v with 0.001v/bit;
		get.SBMU[SBMUcounter].BatteryStatus.ar_CellVoltage[eSubValues.Minimum] := WORD_TO_REAL(DataBuffer[38])/1000;	//0-5v with 0.001v/bit;
		get.SBMU[SBMUcounter].BatteryStatus.ar_CellVoltage[eSubValues.Average] := WORD_TO_REAL(DataBuffer[39])/1000;	//0-5v with 0.001v/bit;
		
		get.SBMU[SBMUcounter].BatteryStatus.ar_CellTemperature[eSubValues.Maximum] := WORD_TO_REAL(DataBuffer[40])-50;	//-50..200gr with 1gr/bit;
		get.SBMU[SBMUcounter].BatteryStatus.ar_CellTemperature[eSubValues.Minimum] := WORD_TO_REAL(DataBuffer[41])-50;	//-50..200gr with 1gr/bit;
		get.SBMU[SBMUcounter].BatteryStatus.ar_CellTemperature[eSubValues.Average] := WORD_TO_REAL(DataBuffer[42])-50;	//-50..200gr with 1gr/bit;
		
		get.SBMU[SBMUcounter].BatteryStatus.r_MaxChargeCurrentAllowed := 		(WORD_TO_REAL(DataBuffer[43])/10)-2000;	//-2k .. +2k A in 0.1A/bit steps
		get.SBMU[SBMUcounter].BatteryStatus.r_MaxDischargeCurrentAllowed := 		(WORD_TO_REAL(DataBuffer[44])/10)-2000;	//-2k .. +2k A in 0.1A/bit steps
		
		get.SBMU[SBMUcounter].BatteryStatus.w_MaxVoltageCellLocation := DataBuffer[48];
		get.SBMU[SBMUcounter].BatteryStatus.w_MinVoltageCellLocation := DataBuffer[49];
		
		get.SBMU[SBMUcounter].BatteryStatus.w_MaxTempCellLocation := DataBuffer[50];
		get.SBMU[SBMUcounter].BatteryStatus.w_MinTempCellLocation := DataBuffer[51];
	
		
		//Collect dataset for CATL datalog
		memcpy(ADR(arDatalogSBMU[SBMUcounter][0]), ADR(DataBuffer[0]), 32); 	//0-15
		tempSBMUStatus.0		:= WORD_TO_BOOL(DataBuffer[16]);
		tempSBMUStatus.1	 	:= WORD_TO_BOOL(DataBuffer[17]);
		tempSBMUStatus.2		:= WORD_TO_BOOL(DataBuffer[18]);
		tempSBMUStatus.3 		:= WORD_TO_BOOL(DataBuffer[19]);
		tempSBMUStatus.4 		:= WORD_TO_BOOL(DataBuffer[20]); 
		tempSBMUStatus.5 		:= WORD_TO_BOOL(DataBuffer[21]);
		arDatalogSBMU[SBMUcounter][16] := tempSBMUStatus;						//16
		memcpy(ADR(arDatalogSBMU[SBMUcounter][17]), ADR(DataBuffer[32]), 44);	//17-38
		arDatalogSBMU[SBMUcounter][39] := DataBuffer[56];						//39
		arDatalogSBMU[SBMUcounter][40] := DataBuffer[57];						//40
		arDatalogSBMU[SBMUcounter][41] := DataBuffer[58];						//41
		arDatalogSBMU[SBMUcounter][42] := DataBuffer[59];						//42
		memcpy(ADR(arDatalogSBMU[SBMUcounter][43]), ADR(DataBuffer[54]), 16);	//43

	(* GIVES RUNTIME EXCEPTION !!! NaN value coming from bms making a runtime exception*)
		//MEMCPY(ADR(get.SBMU[SBMUcounter].BatteryStatus.r_HistAccChargeEnergy), ADR(DataBuffer[85]), 2);  // low word
		//MEMCPY(ADR(get.SBMU[SBMUcounter].BatteryStatus.r_HistAccChargeEnergy)+2, ADR(DataBuffer[84]), 2);  // high word
		//get.SBMU[SBMUcounter].BatteryStatus.r_HistAccChargeEnergy := get.SBMU[SBMUcounter].BatteryStatus.r_HistAccChargeEnergy/10; //0-449GHW with 0.1kWh/bit
		
		//MEMCPY(ADR(get.SBMU[SBMUcounter].BatteryStatus.r_HistAccDischargeEnergy), ADR(DataBuffer[87]), 2);  // low word
		//MEMCPY(ADR(get.SBMU[SBMUcounter].BatteryStatus.r_HistAccDischargeEnergy)+2, ADR(DataBuffer[86]), 2);  // high word
		//get.SBMU[SBMUcounter].BatteryStatus.r_HistAccDischargeEnergy := get.SBMU[SBMUcounter].BatteryStatus.r_HistAccDischargeEnergy/10; //0-449GHW with 0.1kWh/bit
	
		
		get.events.b_SBMUCommError[SBMUCounter] := FALSE;
		
		SBMUCounter := SBMUCounter +1;
		
		IF SBMUCounter >= by_NoOfStrings THEN//BMSGet.MBMU_Status.by_NumberOfSubSystems THEN
			GetSBMUData := TRUE;
			SBMUCounter := 0;
		END_IF
		
		IF 		(get.SBMU[0].b_MainPosRelayClosed AND get.SBMU[0].b_MainNegRelayClosed) OR 
				(get.SBMU[1].b_MainPosRelayClosed AND get.SBMU[1].b_MainNegRelayClosed) OR
				(get.SBMU[2].b_MainPosRelayClosed AND get.SBMU[2].b_MainNegRelayClosed) OR
				(get.SBMU[3].b_MainPosRelayClosed AND get.SBMU[3].b_MainNegRelayClosed) THEN
			PowerStatus := eHVDC_PowerStatus.On;
		ELSIF 	get.SBMU[0].b_PrechargeRelayClosed OR 
				(get.SBMU[1].b_PrechargeRelayClosed AND (by_NoOfStrings > 1)) OR 
				(get.SBMU[2].b_PrechargeRelayClosed AND (by_NoOfStrings > 2))  OR 
				(get.SBMU[3].b_PrechargeRelayClosed AND (by_NoOfStrings > 3)) THEN
			PowerStatus := eHVDC_PowerStatus.Precharging;
		ELSE
			PowerStatus := eHVDC_PowerStatus.Off;
		END_IF	
		
		get.events.b_SBMUFailedToConnect[0] := PowerStatus = eHVDC_PowerStatus.On AND NOT (get.SBMU[0].b_MainPosRelayClosed AND get.SBMU[0].b_MainNegRelayClosed);
		get.events.b_SBMUFailedToConnect[1] := PowerStatus = eHVDC_PowerStatus.On AND (NOT (get.SBMU[1].b_MainPosRelayClosed AND get.SBMU[1].b_MainNegRelayClosed)) AND by_NoOfStrings > 1;
		get.events.b_SBMUFailedToConnect[2] := PowerStatus = eHVDC_PowerStatus.On AND (NOT (get.SBMU[2].b_MainPosRelayClosed AND get.SBMU[2].b_MainNegRelayClosed)) AND by_NoOfStrings > 2;
		get.events.b_SBMUFailedToConnect[3] := PowerStatus = eHVDC_PowerStatus.On AND (NOT (get.SBMU[3].b_MainPosRelayClosed AND get.SBMU[3].b_MainNegRelayClosed)) AND by_NoOfStrings > 3;
		
	ELSE
		get.events.b_SBMUCommError[SBMUCounter] := TRUE;
		SBMUCounter := SBMUCounter +1;
	END_IF
END_IF
END_METHOD

METHOD PRIVATE GetSBMUStaticSystemData : BOOL
VAR_IN_OUT CONSTANT
	st_params			: ST_BMS_params;
END_VAR


VAR_INPUT
	SBMU_ID				:	uint;	
END_VAR

VAR_INST
	MBReadBMS			: 	FB_MBReadRegs;
	DataBuffer 			: 	ARRAY[0..31] OF WORD;
	
	bCommBusy			:	BOOL;
	bComError			:	BOOL;
	errID				:	UDINT;
	cbRead				:	UDINT;
	
	TransmissionDone 	: 	f_trig;
	ComretryCounter		:	USINT := 0;
	
	//ComTimer			:	Ton := (PT := TIME#0S200MS);
END_VAR


VAR
	SBMU: INT;
END_VAR
//Read ETH+MBMU SW/HW version at init.
GetSBMUStaticSystemData := FALSE;

IF (SBMU_ID<1) OR (SBMU>4)then //BMSGET.MBMU_Status.by_NumberOfSubSystems) THEN
	GetSBMUStaticSystemData := TRUE;
	RETURN;
END_IF

ComTimer(in := NOT(ComTimer.Q OR bCommbusy));

MBReadBMS(
sIPAddr := st_params.IP_BMS,
nTCPPort := 502,
nUnitID := 255,//16#FF;
nMBAddr := 960 + (SBMU_ID*1024),
nQuantity := 32,
cbLength := SIZEOF(DataBuffer),
pDestAddr := ADR(DataBuffer),
bExecute := ComTimer.Q,
tTimeout := t_TimeOut,
bBusy => bCommBusy,
bError => bComError,
nErrId => errID,
cbRead => cbRead
);

TransmissionDone(CLK := bCommBusy);

IF TransmissionDone.Q THEN
	IF NOT bComError THEN
	//werkt niet. Bij de MBMU gek genoeg wel
	//	memcpy(destAddr := ADR(BMSGet.SBMU[SBMU_ID].s_SBMU_SWVer), SrcAddr := ADR(DataBuffer[0]), n := 16);
	//	memcpy(destAddr  := ADR(BMSGet.SBMU[SBMU_ID].s_SBMU_HWVer), SrcAddr := ADR(DataBuffer[8]), n := 16);
	//	memcpy(destAddr  := ADR(BMSGet.SBMU[SBMU_ID].s_CSC_SWVer), SrcAddr := ADR(DataBuffer[16]), n := 16);
	//	memcpy(destAddr  := ADR(BMSGet.SBMU[SBMU_ID].s_CSC_HWVer), SrcAddr := ADR(DataBuffer[24]), n := 16);
		GetSBMUStaticSystemData := TRUE;
		get.events.b_SBMUCommError[SBMU_ID] := FALSE;
	ELSE
		get.events.b_SBMUCommError[SBMU_ID] := TRUE;
	END_IF
END_IF
END_METHOD

METHOD PRIVATE GetSystemStatus : BOOL
VAR_IN_OUT CONSTANT
	st_params			: ST_BMS_params;
END_VAR

VAR_INST
	MBReadBMS			: 	FB_MBReadRegs;
	DataBuffer 			: 	ARRAY[0..5] OF WORD;
	
	bCommBusy			:	BOOL;
	bComError			:	BOOL;
	errID				:	UDINT;
	cbRead				:	UDINT;
	
	TransmissionDone 	: 	f_trig;
	
	//ComTimer			:	Ton := (PT := TIME#0S200MS);
	
	ComretryCounter	:	USINT := 0;
END_VAR

//Read general BMS status
GetSystemStatus := FALSE;

ComTimer(in := NOT (ComTimer.Q OR bCommBusy));

MBReadBMS(
sIPAddr := st_params.IP_BMS,
nTCPPort := 502,
nUnitID := 255,//16#FF;
nMBAddr := 769,
nQuantity := 6,
cbLength := SIZEOF(DataBuffer),
pDestAddr := ADR(DataBuffer),
bExecute := ComTimer.Q,
bBusy => bCommBusy,
bError => bComError,
nErrId => errID,
cbRead => cbRead,
tTimeout := t_TimeOut,
);

TransmissionDone(CLK := bCommBusy);

IF TransmissionDone.Q THEN
	IF NOT bComError THEN
		CASE DataBuffer[0] OF
			0: get.MBMU.BatteryStatus.e_BMS_PowerOnStatus := ePowerOnStatus.Off;
			1: get.MBMU.BatteryStatus.e_BMS_PowerOnStatus := ePowerOnStatus.On;
			2: get.MBMU.BatteryStatus.e_BMS_PowerOnStatus := ePowerOnStatus.PowerOn_Fault;
			3: get.MBMU.BatteryStatus.e_BMS_PowerOnStatus := ePowerOnStatus.PowerOff_Fault;
		END_CASE
		
		get.BatteryInfo.e_BMS_PowerOnStatus := get.MBMU.BatteryStatus.e_BMS_PowerOnStatus;
		
		CASE DataBuffer[1] OF
			0: get.MBMU.BatteryStatus.e_BMS_Status := eBMS_Status.Init;
			1: get.MBMU.BatteryStatus.e_BMS_Status := eBMS_Status.Normal;
			2: get.MBMU.BatteryStatus.e_BMS_Status := eBMS_Status.FullCharge;
			3: get.MBMU.BatteryStatus.e_BMS_Status := eBMS_Status.FullDischarge;
			4: get.MBMU.BatteryStatus.e_BMS_Status := eBMS_Status.Warning;
			5: get.MBMU.BatteryStatus.e_BMS_Status := eBMS_Status.Fault;
		END_CASE
		
		get.BatteryInfo.e_BMS_Status := get.MBMU.BatteryStatus.e_BMS_Status;
		
		arDatalogMBMU[48] := DataBuffer[0];
		arDatalogMBMU[49] := DataBuffer[1];
		arDatalogMBMU[50] := DataBuffer[3];
		arDatalogMBMU[51] := DataBuffer[4];
		arDatalogMBMU[52] := DataBuffer[5];	

		
		get.MBMU.by_NumberOfSubSystems := WORD_TO_BYTE(DataBuffer[3]);
		GetSystemStatus := TRUE;
		ComretryCounter := 0;
		b_MBComErrorActive := FALSE;
	ELSE
		COMretryCounter := COMretryCounter +1;
		IF COMRetryCounter > 5 THEN
			b_MBComErrorActive := TRUE;
		END_IF
	END_IF
END_IF
END_METHOD

METHOD GetWearCounters : BOOL
VAR_INST
	PowerOnTimeLogger		:	FB_Varlogger;
	PowerOnCycleLogger		:	FB_Varlogger;
	PrechargeCycleLogger	:	FB_Varlogger;
	OvertempCountLogger		:	FB_Varlogger;
	OverTempTimeLogger		:	FB_Varlogger;
	UnderTempCountLogger	:	FB_Varlogger;
	UnderTempTimeLogger		:	FB_Varlogger;
	
	SlowDataTimer				:	TON := (PT := T#2M);
	rtrig_SOCCalibrationDone	: 	r_trig;
	ton_prechargeDelay			:	ton := (Pt := T#30S);
	
	LastCalibrationTime		:	STRING;
END_VAR
//only log data when BMS communication is actually working
SlowDataTimer(in := NOT SlowDataTimer.q AND BMSDataValid);

PowerOnTimeLogger(		TriggerInput := get.BatteryInfo.e_BMS_PowerOnStatus = ePowerOnStatus.On, 
						LogItemGroup :=  eLogItemGroupID.BMS, 
						LogItemName := 'HVOnHrs', 
						LogType := eLogTypes.TrackOnTime);

PowerOnCycleLogger(		TriggerInput := PowerStatus = eHVDC_PowerStatus.ON, 
						LogItemGroup :=  eLogItemGroupID.BMS, 
						LogItemName := 'HvOnCnt', 
						LogType := eLogTypes.TrackCycles);	

PrechargeCycleLogger(	TriggerInput := PowerStatus = eHVDC_PowerStatus.Precharging, 
						LogItemGroup :=  eLogItemGroupID.BMS, 
						LogItemName := 'PrechargeCnt', 
						LogType := eLogTypes.TrackCycles);	
												
OvertempCountLogger(	TriggerInput := get.Events.b_OVER_TEMP_WARNING, 
						LogItemGroup :=  eLogItemGroupID.BMS, 
						LogItemName := 'OverTempCnt', 
						LogType := eLogTypes.TrackCycles);	

OverTempTimeLogger(		TriggerInput := get.Events.b_OVER_TEMP_WARNING, 
						LogItemGroup :=  eLogItemGroupID.BMS, 
						LogItemName := 'OverTempHrs', 
						LogType := eLogTypes.TrackOnTime);			

UndertempCountLogger(	TriggerInput := get.Events.b_UNDER_TEMP_WARNING, 
						LogItemGroup :=  eLogItemGroupID.BMS, 
						LogItemName := 'UnderTempCnt', 
						LogType := eLogTypes.TrackCycles);	

UnderTempTimeLogger(	TriggerInput := get.Events.b_UNDER_TEMP_WARNING, 
						LogItemGroup :=  eLogItemGroupID.BMS, 
						LogItemName := 'UnderTempHrs', 
						LogType := eLogTypes.TrackOnTime);	

IF BMSDataValid THEN 
	Wearlogging.SetFloat(	eLogItemGroupID.BMS, 	'BattSOH', 				eLogTypes.WriteValue, 			REAL_TO_LREAL(get.BatteryInfo.r_SOH));
	Wearlogging.SetInteger(	eLogItemGroupID.BMS, 	'BattCycles', 			eLogTypes.WriteValue, 			UINT_TO_LINT(get.BatteryInfo.ui_CycleCount));
	Wearlogging.SetFloat(	eLogItemGroupID.BMS, 	'EnergyIn', 			eLogTypes.KeepHighestValue, 	REAL_TO_LREAL(get.BatteryInfo.r_HistAccChargeEnergy));
	Wearlogging.SetFloat(	eLogItemGroupID.BMS, 	'EnergyOut', 			eLogTypes.KeepHighestValue, 	REAL_TO_LREAL(get.BatteryInfo.r_HistAccDischargeEnergy));
	Wearlogging.SetFloat(	eLogItemGroupID.BMS, 	'MaxTempEver', 			eLogTypes.KeepHighestValue, 	REAL_TO_LREAL(get.BatteryInfo.ar_CellTemperature[eSubValues.Maximum]));
	
	IF get.BatteryInfo.ar_CellTemperature[eSubValues.Minimum] > -50 THEN
		Wearlogging.SetFloat(	eLogItemGroupID.BMS, 	'MinTempEver', 			eLogTypes.KeepLowestValue, 		REAL_TO_LREAL(get.BatteryInfo.ar_CellTemperature[eSubValues.Minimum]));
	END_IF
	
	Wearlogging.SetFloat(	eLogItemGroupID.BMS, 	'MaxStringVoltageEver', eLogTypes.KeepHighestValue, 	REAL_TO_LREAL(get.BatteryInfo.r_maxVoltageEver));
END_IF

ton_prechargeDelay(in := get.BatteryInfo.e_BMS_PowerOnStatus = ePowerOnStatus.On);
IF ton_prechargeDelay.Q THEN
	Wearlogging.SetFloat(	eLogItemGroupID.BMS, 	'MinStringVoltageEver', 		eLogTypes.KeepLowestValue, 	REAL_TO_LREAL(get.BatteryInfo.r_SystemVoltage));
END_IF


rtrig_SOCCalibrationDone(clk := get.BatteryInfo.e_BMS_Status = eBMS_Status.FullCharge);		
IF rtrig_SOCCalibrationDone.Q THEN
	dt_LastCalibrationDate := gvl.dt_SystemDateTime;
	LastCalibrationTime:= DT_TO_STRING(gvl.dt_SystemDateTime);
	Wearlogging.SetString(eLogItemGroupID.BMS, 'LastSocCalibration', 	LastCalibrationTime);
END_IF

IF slowDataTimer.Q THEN
	slowDataTimer.Q;
END_IF
							
//Add: Last calibration date
END_METHOD

METHOD Init : BOOL
VAR_INPUT
END_VAR

VAR
	temp1	:	LREAL;
	temp2	:	LREAL;
END_VAR
IF NOT InitDone THEN
	Wearlogging.GetFloatValue(eLogItemGroupID.BMS, 	'EnergyIn', CurrentLogValue => temp1);
	get.BatteryInfo.r_HistAccDischargeEnergy := LREAL_TO_REAL(temp1);
	get.MBMU.BatteryStatus.r_HistAccDischargeEnergy := LREAL_TO_REAL(temp1);
	
	Wearlogging.GetFloatValue(eLogItemGroupID.BMS, 	'EnergyOut', CurrentLogValue => temp2);
	
	get.BatteryInfo.r_HistAccChargeEnergy := LREAL_TO_REAL(temp2);
	get.MBMU.BatteryStatus.r_HistAccChargeEnergy := LREAL_TO_REAL(temp2);

	Wearlogging.SetInteger(	eLogItemGroupID.BMS, 	'nameplateEnergyCapacity', 			eLogTypes.WriteValue, 			REAL_TO_LINT(Settings.Properties.r_RatedEnergyCapacity));
	InitDone := TRUE;
END_IF
END_METHOD

METHOD PRIVATE OpenInsulationSwitch : BOOL
VAR_IN_OUT CONSTANT
	st_params			: ST_BMS_params;
END_VAR

VAR_INPUT
	OpenSwitch : BOOL;
END_VAR

VAR_INST
	WriteReg	:	FB_MBWriteSingleReg;
	Value 		:	WORD 	:= 0;
	StartWrite	:	BOOL	:= FALSE;
	
	bCommBusy	:	BOOL;
	bComError	:	BOOL;
	errID		:	UDINT;

	TransmissionDone 	: 	f_trig;
	ComRetryCounter	:	USINT;
	
	ComTimer			:	Ton := (PT := TIME#0S200MS);
END_VAR

ComTimer(in := NOT(ComTimer.Q));

OpenInsulationswitch := FALSE;

IF OpenSwitch THEN
	Value := 1;
ELSE
	Value := 0;
END_IF

WriteReg(
sIPAddr := st_params.IP_BMS,
nTCPPort := 502,
nUnitID := 255,//16#FF;
nMBAddr := 907,
nValue := Value,
tTimeout := T#0S100MS,
bExecute := ComTimer.q,
bBusy => bCommBusy,
bError => bComError,
nErrId => errID,
);

TransmissionDone(CLK := bCommBusy);

IF TransmissionDone.Q THEN
	IF NOT bComError THEN
		arDatalogEMS[3] := 1;	
		get.MBMU.b_InsulationSwitchOpen := OpenSwitch;
		ComRetryCounter := 0;
		OpenInsulationSwitch := TRUE;
		b_MBComErrorActive := FALSE;
	ELSE
		COMretryCounter := COMretryCounter +1;
		IF COMRetryCounter > 5 THEN
			b_MBComErrorActive := TRUE;
		END_IF
	END_IF
END_IF
END_METHOD

METHOD Reset : BOOL
VAR_INPUT
	//BMSSET	:	st_BMS_Set;
	//ResetIn	:	BOOL;
END_VAR

VAR_INST
	ResetTrigger		:	Ton := (PT := TIME#1S0MS);
	ResetVar			:	BOOL;
END_VAR
b_MBComErrorActive := FALSE;
Reset := ClearBMSFaults(st_params);

FBState := ePOUState.Normal;
END_METHOD

METHOD PRIVATE SetBMSDateTime : BOOL
VAR_IN_OUT CONSTANT
	st_params			: ST_BMS_params;
END_VAR

VAR
	SystemTimeData	:	Timestruct;
	RTCData	:	ARRAY[0..6] OF WORD;	
	
END_VAR
VAR_INST
	//ComTimer			:	Ton := (PT := TIME#0S200MS);
	WriteRegs		:	FB_MBWriteRegs;
	SystemTime		:	FB_LocalSystemTime;
	TransmissionDone 	: 	f_trig;
	SystemTimeDataValid	:	BOOL;
	bCommBusy		:	BOOL;
	bComError		:	BOOL;
	errID			:	UDINT;
	COMRetryCounter	:	USINT := 0;
END_VAR
ComTimer(in := NOT(ComTimer.Q OR bCommBusy));

//write PLC system time to BMS RTC
SetBMSDateTime := FALSE;


//retrieve system time struct
SystemTime(
	sNetID := '',
	bEnable := TRUE,
	dwCycle := 1,
	dwOpt	:= 1,
	tTimeout := t_TimeOut,
	bValid => SystemtimeDataValid,
	systemTime => SystemTimeData
);

//parse system time to BMS data array
IF SystemTimeDataValid THEN
	RTCData[0] := 2024;//SystemTimeData.wYear;
	RTCData[1] := 03;//SystemTimeData.wMonth;
	RTCData[2] := 26;//SystemTimeData.wDay;
	RTCData[3] := 13;//SystemTimeData.wHour;
	RTCData[4] := 52;//SystemTimeData.wMinute;
	RTCData[5] := 00;//SystemTimeData.wSecond;
	RTCData[6] := 1;//can this value remain at 1? or reset to 0 after write?
	
	//write data to BMS
	WriteRegs(	
	sIPAddr := st_params.IP_BMS,
	nTCPPort := 502,
	nUnitID := 255,//16#FF;
	nMBAddr := 900,
	nQuantity := 7,
	pSrcAddr := ADR(RTCData),
	cbLength := SIZEOF(RTCData),
	bExecute := ComTimer.Q,
	tTimeout := TIME#100MS,
	bBusy => bCommBusy,
	bError => bComError,
	nErrId => errID,
	);
	
	TransmissionDone(CLK := bCommBusy);
	
	//return true if tranmission succeeds
	IF TransmissionDone.Q THEN
		IF NOT bComError THEN
			SetBMSDateTime := TRUE;
			ComRetryCounter := 0;
			b_MBComErrorActive := FALSE;
		ELSE
			COMretryCounter := COMretryCounter +1;
			IF COMRetryCounter > 5 THEN
				b_MBComErrorActive := TRUE;
			END_IF
		END_IF
	END_IF
END_IF
END_METHOD

METHOD PRIVATE SetPowerMode : BOOL
VAR_IN_OUT CONSTANT
	st_params			: ST_BMS_params;
END_VAR

VAR_INST
	WriteReg	:	FB_MBWriteSingleReg;
	Value 		:	WORD 	:= 1;
	StartWrite	:	BOOL	:= FALSE;
	bCommBusy	:	BOOL;
	bComError	:	BOOL;
	errID		:	UDINT;
	TransmissionDone 	: 	f_trig;
	//ComTrigger	:	Ton := (PT := TIME#200MS);
	ComRetryCounter	:	USINT	:= 0;
	
	b_HVRequest			: BOOL;
	ton_StartRetrigger	: ton :=(PT := T#5S);
END_VAR	

VAR_INST
	rtrigPowerOn		: R_trig;
END_VAR

//Value := ePowerControl.Stay; //default command is: Do nothing
//it may also work if we just keep sending "poweron" if b_HVDC_Required is true. But this doesn't seem to be the way they intended.
b_HVRequest := b_HVDC_OnRq AND NOT ton_StartRetrigger.Q AND get.BatteryInfo.e_BMS_PowerOnStatus <> ePowerOnSTatus.On;
ton_StartRetrigger(IN:=b_HVRequest);
rtrigPowerOn(CLK:= ton_StartRetrigger.Q);



IF NOT b_HVDC_OnRq AND get.BatteryInfo.e_BMS_PowerOnStatus <> ePowerOnSTatus.Off THEN
	Value := ePowerControl.PowerOff;
ELSIF rtrigPowerOn.Q THEN
	Value := ePowerControl.PowerOn;
END_IF

//Write this register every second, regardless of change.
ComTimer(in := NOT(ComTimer.Q OR bCommBusy));

//IF BMSGet.BattInfo.ui_BMS_Status < 5 THEN
WriteReg(
	sIPAddr := st_params.IP_BMS,
	nTCPPort := 502,
	nUnitID := 255,//16#FF;
	nMBAddr := 897,
	nValue := Value,
	tTimeout := t_TimeOut,
	bExecute := ComTimer.Q,
	bBusy => bCommBusy,
	bError => bComError,
	nErrId => errID,
);
//ELSE
//	SetPowerMode := TRUE;
//END_IF

TransmissionDone(CLK := bCommBusy);
	
//return true if tranmission succeeds
IF TransmissionDone.Q THEN
	IF NOT bComError THEN
		arDatalogEMS[1] := Value;	
	
		SetPowerMode := TRUE;
		ComRetryCounter := 0;
		Value := ePowerControl.Stay;
		b_MBComErrorActive := FALSE;
	ELSE
		COMretryCounter := COMretryCounter +1;
		IF COMRetryCounter > 5 THEN
			b_MBComErrorActive := TRUE;
		END_IF
	END_IF
END_IF
END_METHOD

ACTION SFCTipReset:
SFCTip := FALSE;
END_ACTION

END_FUNCTION_BLOCK

// ---- POUs/Objects/BMS/FB_BMS_IO.TcPOU
FUNCTION_BLOCK FB_BMS_IO

VAR_INPUT
	b_BMSEnable			 AT %Q* : BOOL;
END_VAR

END_FUNCTION_BLOCK

// ---- POUs/Functions-FBs-Programs/_generalFunctions/F_RoundReal.TcPOU
FUNCTION F_RoundReal : REAL
VAR_INPUT
  rInput : REAL;
  iDecimalPlaces : INT;
END_VAR
VAR
  rOutput : REAL;
  r_Dint: DINT;
  rLeftPart : REAL;
END_VAR

rOutput := rInput * EXPT(10, iDecimalPlaces);
rLeftPart := rOutput - TRUNC(rOutput);

rOutput := TRUNC(rOutput);

IF rLeftPart >= 0.5 THEN
  	rOutput:= rOutput + 1;
ELSE
  	rOutput := rOutput;
END_IF

F_RoundReal := rOutput / EXPT(10, iDecimalPlaces);

END_FUNCTION

// ---- POUs/Objects/ProtectionSystems/FB_ProtectionSystems.TcPOU
FUNCTION_BLOCK FB_ProtectionSystems
VAR_IN_OUT CONSTANT
	st_params				: ST_Protectionsystems_params;
END_VAR

VAR_OUTPUT
	get						: ST_ProtectionSystems_get;
	b_SystemShutdownCMD		: BOOL;
END_VAR

VAR_INPUT
	set						: ST_ProtectionSystems_set;
	
	b_BatteryAlarm			: BOOL;
END_VAR

VAR_IN_OUT CONSTANT
	Powermonitor : st_powermonitor_get;
END_VAR

VAR
	Firedetection			: FB_Firedetection;
	InsulationMonitor		: FB_InsulationMonitor;
	SurgeProtection			: FB_SurgeProtection;
	ResidualCurrentMonitor	: FB_RCmonitor;
	OverCurrentProtection	: FB_OvercurrentProtection;
END_VAR

VAR_INPUT
	ToInsuMon				:	St_InsulationMonitor_PassThrough;
END_VAR

firedetection(st_params := st_params.firedetection, get => get.FireDetection, set := set.FireDetection, b_SystemShutdownCMD => b_systemshutdownCMD, b_batteryAlarm:= b_batteryalarm);

InsulationMonitor(ToInsuMon := ToInsuMon, get => get.Insulation, set := set.Insulation,
st_params := st_params.InsulationMonitor);

SurgeProtection(get => get.Surge);

ResidualCurrentMonitor(get => get.MRCDB);

OverCurrentProtection(st_params := st_Params.OCP,
	get=>get.OvercurrentProtection,
	powermonitor := powermonitor,
	set:= set.OvercurrentProtection,
	b_inputsectionAvailable := settings.Configuration.b_ACInputConnection,
	b_thirdOutputAvailable := settings.configuration.b_ThirdOutputConnection);

METHOD GetDiagnostics
VAR_IN_OUT
	AddError		: ARRAY [*] OF FB_AddErrorST;
	a_ActiveEvents	: ARRAY [*] OF ST_ErrorStruct;
	w_Index			: WORD;
END_VAR
Firedetection.GetDiagnostics(Adderror := AddError, a_ActiveEvents := a_ActiveEvents, w_Index := w_index);
Surgeprotection.GetDiagnostics(Adderror := AddError, a_ActiveEvents := a_ActiveEvents, w_Index := w_index);
InsulationMonitor.GetDiagnostics(Adderror := AddError, a_ActiveEvents := a_ActiveEvents, w_Index := w_index);
ResidualCurrentMonitor.GetDiagnostics(Adderror := AddError, a_ActiveEvents := a_ActiveEvents, w_Index := w_index);
OvercurrentProtection.GetDiagnostics(Adderror := AddError, a_ActiveEvents := a_ActiveEvents, w_Index := w_index);
END_METHOD

METHOD PUBLIC Reset : BOOL
VAR_INPUT
END_VAR
Reset := Firedetection.Reset() AND OvercurrentProtection.Reset() AND insulationmonitor.Reset() AND ResidualCurrentMonitor.Reset();
END_METHOD

END_FUNCTION_BLOCK

// ---- POUs/Objects/ProtectionSystems/FireDetection/FB_FireDetection.TcPOU
FUNCTION_BLOCK FB_FireDetection
VAR_IN_OUT CONSTANT
	st_params	: ST_Firedetection_params;
END_VAR

VAR_OUTPUT
	get						:	ST_FireDetection_get;
END_VAR

VAR_OUTPUT	
	b_SystemShutdownCMD 	: 	BOOL;
END_VAR

VAR_INPUT
	Set						:	ST_FireDetection_Set;
	b_BatteryAlarm			: 	BOOL;
END_VAR

VAR	
	b_FireAlarm				: 	BOOL;
	ton_ShutdownDelay		: 	TON := (PT := T#10S);
	ton_SounderOffReset		: 	TON := (PT := T#1S);
	SmokeDetPowerDownTimer 	: 	TP := (PT := TIME#500MS);
END_VAR

VAR
	IO								: FB_FireDetection_IO;
END_VAR

VAR CONSTANT
	w_ID							: WORD := eObject_ID.FireDetection;
END_VAR

IO(st_params:= st_params);

CheckSmokeDetectors(get.SmokeDetectors);
CheckCODetectors(st_params, get.CODetectors);
SounderBeacon();
SetEvents();

get.b_FireAlarm := (get.CODetectors.State = eCOAlarmStatus.Alarm OR get.SmokeDetectors.State = eSmokeDetectAlarmStatus.Alarm);
ton_ShutdownDelay(IN:= b_BatteryAlarm AND get.b_FireAlarm);
IF ton_ShutdownDelay.Q THEN
	b_SystemShutdownCMD := TRUE;
END_IF

//Smoke detector reset
SmokeDetPowerDownTimer(Q => io.SmokeDetectorOFF);
SmokeDetPowerDownTimer.IN := FALSE;

ton_SounderOffReset(IN:= io.SounderOFF);
IF ton_SounderOffReset.Q THEN
	io.SounderOFF := FALSE;
END_IF

METHOD PRIVATE CheckCODetectors : BOOL
VAR_IN_OUT CONSTANT
	st_params : ST_Firedetection_params;
END_VAR

VAR_IN_OUT
	data			: ST_CODetectors;
END_VAR

VAR_INST
	Warning1Timer	:	TON := (PT := TIME#60S);
	Warning2Timer	:	TON := (PT := TIME#60S);
	ErrorTimer		:	TON := (PT := TIME#10S);	
	b_test			:	BOOL; 
END_VAR

VAR
	CoLevelMean			: REAL;
END_VAR
//actual sensor value already filled in in IO code. Only generate status data here.
//alarm status can not be cleared in this method. only via fb_firedetection.reset method.
//alarm status is te highest status, if true, no work to do here.
//if both sensors are working
CoLevelMean := (io.CODetector[1] + io.CODetector[2]) / 2;
data.Value[0] := SEL(CoLevelMean > 5, CoLevelMean, 0);
data.Value[1] := io.CODetector[1];
data.Value[2] := io.CODetector[2];
data.Value[3] := MAX(io.CODetector[1],io.CODetector[2]);

ErrorTimer		(IN := CoLevelMean > st_params.r_COalarmLevel);
Warning1Timer	(IN := CoLevelMean > st_params.r_COwarningLevel_1);
Warning2Timer	(IN := CoLevelMean > st_params.r_COwarningLevel_2);
	
//sr_COalarmState(Set1:=ErrorTimer.Q OR b_test);
//sr_COalarmState.RESET := FALSE;

IF ErrorTimer.Q THEN
	data.State := eCOAlarmStatus.Alarm;
END_IF
	
IF data.State <> eCOAlarmStatus.Alarm THEN
	IF Warning2Timer.Q THEN
		data.State := eCOAlarmStatus.WarningLevel2;
	ELSIF Warning1Timer.Q THEN
		data.State := eCOAlarmStatus.WarningLevel1;
	ELSIF (io.CODetector[1] = -1) OR (io.CODetector[2] = -1) THEN
		data.State := eCOAlarmStatus.Error;
	ELSE
		data.State := eCOAlarmStatus.Normal;
	END_IF
END_IF

data.b_CoValuesOK := NOT (ErrorTimer.Q OR data.State = eCOAlarmStatus.Error);
END_METHOD

METHOD PRIVATE CheckSmokeDetectors

VAR_IN_OUT
	data : ST_Smokedetectors;
END_VAR

VAR_INST
	AlarmResetTimer: TP := (PT := TIME#500MS);
	SmokeAlarmTimer: TON := (PT := TIME#500ms);
	AlarmResetTrigger: F_TRIG;
	SmokeAlarmPowerLost: TON := (PT := TIME#50MS);
END_VAR
//input delay for alarm inputs
SmokeAlarmTimer(IN := (NOT io.SmokeDetector.Signal_OK) AND (NOT AlarmResetTrigger.Q));
SmokeAlarmPowerLost(IN := (NOT  io.SmokeDetector.Power_OK) AND  (NOT AlarmResetTrigger.Q));

IF data.State = eSmokeDetectAlarmStatus.Normal THEN
	IF SmokeAlarmPowerLost.Q THEN	//Alarm power failure means alarm cannot be trusted. So first check power
		data.State := eSmokeDetectAlarmStatus.Error;
	ELSIF SmokeAlarmTimer.Q THEN	//if alarm signals for >500ms --> raise the alarm.
		data.State := eSmokeDetectAlarmStatus.Alarm;	//alarm is only resettable manually via resetDetectors
	END_IF
ELSIF get.SmokeDetectors.State = eSmokeDetectAlarmStatus.Error THEN	//if power failed, no alarm checking anymore as this will give false alarms
	IF NOT SmokeAlarmPowerLost.Q THEN	//Alarm state may return to operational if power comes back
		data.State := eSmokeDetectAlarmStatus.Normal;
	END_IF
END_IF	//In alarm state, no power checking is performed anymore. Even if the detectors lose power now, the alarm state has priority.
END_METHOD

METHOD PUBLIC EMstop : BOOL
VAR_INPUT
END_VAR
//do anything?
//return true when ready
END_METHOD

METHOD GetDiagnostics
VAR_IN_OUT
	AddError		: ARRAY [*] OF FB_AddErrorST;
	a_ActiveEvents	: ARRAY [*] OF ST_ErrorStruct;
	w_Index			: WORD;
END_VAR
(*Alarm Muted *)		AddError[w_Index](
		b_ErrorTrig			:= get.events.AlarmMuted,
		out_ST_Error			:= a_ActiveEvents[w_Index],
		w_ErrorID					:= 1,
		e_ObjectID				:= eObject_ID.Firedetection,
		s_Message				:= 'alarm muted',
		e_sev					:= eseverity.info,
		b_AutoClear				:= TRUE,
		e_ErrAckAccess		:= eErrAckAccess.General
	);
	w_Index := w_Index +1;

(*Smoke NOK*)			AddError[w_Index](
		b_ErrorTrig			:= get.events.SmokeDetFault,
		out_ST_Error			:= a_ActiveEvents[w_Index],
		w_ErrorID					:= 2,
		s_Message				:= 'smoke detector not OK',
		e_sev					:= eseverity.warning,
		t_triggerTime			:= T#5S,
		b_AutoClear				:= TRUE,
		e_ErrAckAccess		:= eErrAckAccess.operator,
	);
	w_Index := w_Index +1;

(*Smoke alarm*)			AddError[w_Index](
		b_ErrorTrig				:= get.events.SmokeDetAlarm,
		out_ST_Error			:= a_ActiveEvents[w_Index],
		w_ErrorID				:= 3,
		s_Message				:= 'smoke detector alarm',
		e_sev					:= eseverity.Quickshutdown,
		e_ErrAckAccess			:= eErrAckAccess.VDL,
		b_SMSEnableVDL			:= TRUE,
	);
	w_Index := w_Index +1;

(*CO NOK*)				AddError[w_Index](
		b_ErrorTrig				:= get.events.CODetFault,
		out_ST_Error			:= a_ActiveEvents[w_Index],
		w_ErrorID				:= 4,
		s_Message				:= 'CO detector not OK',
		e_sev					:= eseverity.Warning,
		b_AutoClear				:= TRUE,
		e_ErrAckAccess			:= eErrAckAccess.operator,
		t_TriggerTime			:= T#2S,
	);
	w_Index := w_Index +1;

(*CO warning level1*)			AddError[w_Index](
		b_ErrorTrig				:= get.events.CODetWarning1,
		out_ST_Error			:= a_ActiveEvents[w_Index],
		w_ErrorID				:= 5,
		s_Message				:= CONCAT(CONCAT('CO Detector warning level 1: ', TO_STRING(st_params.r_COwarningLevel_1)), ' ppm'),
		e_sev					:= eseverity.info,
		e_ErrAckAccess			:= eErrAckAccess.Operator,
		b_AutoClear				:= TRUE,
		b_SMSEnableVDL			:= FALSE,
	);
	w_Index := w_Index +1;
	
(*CO warning level2*)			AddError[w_Index](
		b_ErrorTrig				:= get.events.CODetWarning2,
		out_ST_Error			:= a_ActiveEvents[w_Index],
		w_ErrorID				:= 6,
		s_Message				:= CONCAT(CONCAT('CO Detector warning level 2: ', TO_STRING(st_params.r_COwarningLevel_2)), ' ppm'),
		e_sev					:= eseverity.Warning,
		e_ErrAckAccess			:= eErrAckAccess.operator,
		b_AutoClear				:= TRUE,
		b_SMSEnableVDL			:= FALSE,
	);
	w_Index := w_Index +1;

(*CO alarm*)			AddError[w_Index](
		b_ErrorTrig				:= get.events.CODetAlarm,
		out_ST_Error			:= a_ActiveEvents[w_Index],
		w_ErrorID				:= 7,
		s_Message				:=  CONCAT(CONCAT('CO Detector alarm level: ', TO_STRING(st_params.r_COAlarmLevel)), ' ppm'),
		e_sev					:= eseverity.NormalShutdown,
		e_ErrAckAccess			:= eErrAckAccess.VDL,
		b_SMSEnableVDL			:= TRUE,
	);
	w_Index := w_Index +1;
END_METHOD

METHOD PUBLIC Reset : BOOL
VAR_INPUT
//	ResetActive : BOOL := FALSE;
END_VAR

VAR_INST
	b_status : BOOL;
END_VAR
//return true when ready



IF io.smokedetector.Power_OK AND io.smokedetector.Signal_OK THEN
	get.SmokeDetectors.State := eSmokeDetectAlarmStatus.Normal;
END_IF

IF get.CODetectors.b_CoValuesOK THEN
	get.CODetectors.State := eCOAlarmStatus.Normal;
END_IF

b_status := get.CODetectors.State = eCOAlarmStatus.Normal AND get.SmokeDetectors.State = eSmokeDetectAlarmStatus.Normal;
SmokeDetPowerDownTimer.IN := NOT b_status;

IF b_status THEN
	io.SounderON := FALSE;
	io.SounderOFF := TRUE;
END_IF

Reset := b_status AND io.smokedetector.Power_OK;
END_METHOD

METHOD SetEvents : BOOL
VAR_INPUT
END_VAR
get.Events.SmokeDetAlarm 	:= (get.SmokeDetectors.State = eSmokeDetectAlarmStatus.Alarm);
get.Events.SmokeDetFault 	:= (get.SmokeDetectors.State = eSmokeDetectAlarmStatus.Error);
get.Events.CODetAlarm 		:= (get.CODetectors.State = eCOAlarmStatus.Alarm);
get.Events.CODetFault 		:= (get.CODetectors.State = eCOAlarmStatus.Error);
get.Events.CODetWarning1	:= get.CODetectors.State = eCOAlarmStatus.WarningLevel1;
get.Events.CODetWarning2	:= get.CODetectors.State = eCOAlarmStatus.WarningLevel2;

get.Events.AlarmMuted 		:= (get.Events.SmokeDetAlarm OR get.Events.CODetAlarm) And not io.SounderOn;
END_METHOD

METHOD SounderBeacon : BOOL

VAR_INST
	
	TestTrigger 		: 	R_Trig;
	SmokeAlarmTrigger	:	R_Trig;
	COAlarmTrigger		:	R_trig;
END_VAR

//Only enable sounder at the start of the alarm. Use old_state to determine this.
//This allows for alarm muting and retriggering. 
COAlarmTrigger(clk:=get.CODetectors.State = eCOAlarmStatus.Alarm);
SmokeAlarmTrigger(Clk:= get.SmokeDetectors.State = eSmokeDetectAlarmStatus.Alarm);

//use rtrig to prevent permanent sounding. resilence with muting.
TestTrigger(clk:= set.TestSounder);

//use rtrig to prevent permanent muting.
IF set.SilenceSounder THEN
	io.SounderOn:= FALSE;
	io.SounderOFF := TRUE;
END_IF

IF COAlarmTrigger.q OR SmokeAlarmTrigger.Q OR TestTrigger.Q THEN;
	io.SounderOn:= TRUE;
END_IF
END_METHOD

END_FUNCTION_BLOCK

// ---- POUs/Objects/ProtectionSystems/FireDetection/FB_FireDetection_IO.TcPOU
FUNCTION_BLOCK FB_FireDetection_IO

VAR_IN_OUT CONSTANT
	st_params				: ST_Firedetection_params;
END_VAR

VAR
	CO_read							AT %I*	: ARRAY [1..2] OF ST_AnalogInputData;
END_VAR

VAR_OUTPUT
	SmokeDetector					AT %I*	:	ST_SmokeDetIO;
	CODetector								:	ARRAY[1..2] OF REAL;
END_VAR

VAR_INPUT
	SounderON						AT %Q* 	: BOOL;	
	SounderOFF						AT %Q* 	: BOOL;
	SmokeDetectorOFF				AT %Q* 	: BOOL;
END_VAR

CO_detector_IO();

METHOD CO_detector_IO : BOOL
IF CO_read[1].Status.Overrange OR CO_read[1].Status.Underrange THEN
	CODetector[1] := -1;
ELSE
	CODetector[1] := scale(CO_read[1].Value, In_min := 0, In_Max := 16#8000, Out_min:= 0, Out_max:= st_params.r_COrange);
END_IF

IF CO_read[2].Status.Overrange OR CO_read[2].Status.Underrange THEN
	CODetector[2] := -1;
ELSE
	CODetector[2] := scale(CO_read[2].Value, In_min := 0, In_Max := 16#8000, Out_min:= 0, Out_max:= st_params.r_COrange);
END_IF
END_METHOD

END_FUNCTION_BLOCK

// ---- POUs/Objects/ProtectionSystems/InsulationMonitoring/FB_InsulationMonitor.TcPOU
FUNCTION_BLOCK FB_InsulationMonitor

VAR_OUTPUT
	get			: ST_InsulationMonitor_get;
END_VAR

VAR_INPUT
	set			: ST_InsulationMonitor_set;
END_VAR

VAR_IN_OUT
	ToInsuMon			: St_InsulationMonitor_PassThrough;
END_VAR

VAR_IN_OUT CONSTANT
	st_params			: St_InsulationMonitor_params;
END_VAR

VAR CONSTANT
	w_ID			: WORD := eObject_ID.InsulationMonitor;
END_VAR

VAR
	t_DisableTime						: TIME;
	b_SystemConnected					: BOOL;
	b_disablecondition					: BOOL;
	b_PENlinkDiscrepance				: BOOL;
	b_prewarningOK				AT %I* : BOOL;
	b_DisableInsulationTrip		AT %Q* : BOOL;
	
	rtrig_InsulationDisable		: R_TRIG;
	sr_TripDisable				: SR;
	ton_EvaluationTime			: TON := (PT:=T#10S);
	ton_disableOffDelay			: TON := (PT:=T#10S);
	
	b_PenStateLast					: BOOL;			
END_VAR

get.b_Warning := FALSE;
get.b_NoEarthingSystemSet := set.e_EarthingSystem = eEarthingSystems.None;
b_SystemConnected := (ToInsuMon.b_MccbfbMaster OR ToInsuMon.b_MccbfbSlave) AND ToInsuMon.b_NetContFB;
b_disableCondition:= set.e_EarthingSystem = eEarthingSystems.TN;

IF NOT b_disableCondition THEN
	get.b_Warning := NOT(b_prewarningOK);
END_IF

//trigger when pen link is switched during operation, resulting in an quickshutdown.
//IF ToInsuMon.b_NetContFB AND b_PenStateLast <> toInsuMon.b_PENlinkFB THEN
//	get.b_PENlinkOperatedFault := TRUE;
//ELSE
//	b_PenStateLast := toInsuMon.b_PENlinkFB;
//END_IF
t_DisableTime:=  TO_TIME(st_params.i_EarthSystemDetectionDelay * 1000);
//when isolation monitor needs re-enabled
ton_disableOffDelay(IN:= NOT b_SystemConnected, PT := t_DisableTime);

// On netcontactor in trigger
ton_EvaluationTime(IN:= b_SystemConnected AND b_prewarningOK, PT :=t_DisableTime);
rTrig_InsulationDisable(CLK:= b_SystemConnected AND b_disableCondition);

//if no warning shows up during disabled monitor, it means that PE-Neutral link is NOT properly made in the network.
sr_TripDisable(SET1:= rTrig_insulationDisable.Q, Q1=> b_disableInsulationTrip);
sr_TripDisable.RESET := ton_EvaluationTime.Q OR ton_disableOffDelay.Q; //so reactivate trip when no warning is detected



IF b_SystemConnected AND b_disablecondition THEN
	IF sr_TripDisable.Q1 THEN
		get.e_EarthingSystemDetected := set.e_EarthingSystem;
		get.b_PENlinkDetected := TRUE;
		b_PENlinkDiscrepance := FALSE;
	ELSIF ton_EvaluationTime.Q THEN
		b_PENlinkDiscrepance := TRUE;
	END_IF
	
ELSE
	get.e_EarthingSystemDetected := eEarthingsystems.IT;
	get.b_PENlinkDetected := FALSE;
	b_PENlinkDiscrepance := FALSE;
END_IF

//if IT is configured and PEN is connected in system, raise error beforehand.
get.b_EarthingSystemMismatch := ToInsuMon.b_PENlinkFB AND set.e_EarthingSystem = eEarthingSystems.IT;

//Couple gets
get.b_Enabled := NOT(b_disableInsulationTrip);

METHOD GetDiagnostics
VAR_IN_OUT
	AddError		: ARRAY [*] OF FB_AddErrorST;
	a_ActiveEvents	: ARRAY [*] OF ST_ErrorStruct;
	w_Index			: WORD;
END_VAR

VAR_INST
	index : WORD;
END_VAR
index := w_index;

(*Disabled message*)			AddError[w_Index](
		b_ErrorTrig			:= NOT(get.b_Enabled),
		out_ST_Error			:= a_ActiveEvents[w_Index],
		w_ErrorID					:= 1,
		e_ObjectID				:= eObject_ID.InsulationMonitor,
		s_Message				:= 'disabled',
		e_sev					:= eseverity.info,
		b_AutoClear			:= TRUE
	);
	w_Index := w_Index +1;

(*warning*)			AddError[w_Index](
		b_ErrorTrig			:= get.b_warning,
		out_ST_Error			:= a_ActiveEvents[w_Index],
		w_ErrorID					:= 2,
		s_Message				:= 'warning level',
		e_sev					:= eseverity.warning,
		e_ErrAckAccess		:= eErrAckAccess.operator
	);
	w_Index := w_Index +1;
	
(*PEN link detected*)			AddError[w_Index](
		b_ErrorTrig			:= get.b_PENlinkDetected,
		out_ST_Error			:= a_ActiveEvents[w_Index],
		w_ErrorID					:= 3,
		s_Message				:= 'PEN link detected',
		e_sev					:= eseverity.info,
		e_ErrAckAccess		:= eErrAckAccess.operator,
		b_autoClear			:= TRUE
	);
	w_Index := w_Index +1;
	
(*PENlinkmissing*)			AddError[w_Index](
		b_ErrorTrig			:= b_PENlinkdiscrepance,
		out_ST_Error			:= a_ActiveEvents[w_Index],
		w_ErrorID					:= 4,
		s_Message				:= 'PEN link not detected in TN earthing system',
		e_sev					:= eseverity.NormalShutdown,
		e_ErrAckAccess		:= eErrAckAccess.operator
	);
	w_Index := w_Index +1;
	
(*PENlink operated during operation*)			AddError[w_Index](
		b_ErrorTrig			:= get.b_PENlinkOperatedFault,
		out_ST_Error			:= a_ActiveEvents[w_Index],
		w_ErrorID					:= 5,
		s_Message				:= 'PEN link switched during operation',
		e_sev					:= eseverity.Warning,  //eseverity.NormalShutdown,
		e_ErrAckAccess		:= eErrAckAccess.operator
	);
	w_Index := w_Index +1;
(*Earthing system mismatch*)			AddError[w_Index](
		b_ErrorTrig			:= get.b_EarthingSystemMismatch,
		out_ST_Error			:= a_ActiveEvents[w_Index],
		w_ErrorID					:= 6,
		s_Message				:= 'Configured earthing system not corresponding to PENlink state',
		e_sev					:= eseverity.Normalshutdown,
		e_ErrAckAccess		:= eErrAckAccess.operator
	);
	w_Index := w_Index +1;
	
(*Earthing system mismatch*)			AddError[w_Index](
		b_ErrorTrig			:= get.b_NoEarthingSystemSet,
		out_ST_Error			:= a_ActiveEvents[w_Index],
		w_ErrorID					:= 7,
		s_Message				:= 'No earthing system select, starting not allowed',
		e_sev					:= eseverity.warning,
		b_AutoClear			:= TRUE
	);
	w_Index := w_Index +1;
END_METHOD

METHOD Reset : BOOL
VAR_INPUT
END_VAR
b_penlinkdiscrepance := FALSE;
get.b_PENlinkOperatedFault := FALSE;

Reset := b_prewarningOK AND NOT(get.b_PENlinkOperatedFault OR b_penlinkdiscrepance);
END_METHOD

END_FUNCTION_BLOCK

// ---- POUs/Objects/ProtectionSystems/SurgeProtection/FB_SurgeProtection.TcPOU
FUNCTION_BLOCK FB_SurgeProtection
VAR_OUTPUT
	get				: ST_surgeprotection_get;
END_VAR

VAR CONSTANT
	w_ID			: WORD := eObject_ID.SurgeProtection;
END_VAR

VAR	
	
	a_bRead					AT %I* : ARRAY [1..2] OF BOOL;
END_VAR

get.b_Type12_OK := a_bRead[2];
get.b_Type3_OK 	:= a_bRead[1];

METHOD GetDiagnostics
VAR_IN_OUT
	AddError		: ARRAY [*] OF FB_AddErrorST;
	a_ActiveEvents	: ARRAY [*] OF ST_ErrorStruct;
	w_Index			: WORD;
END_VAR
(*Type1/2 warning*)			AddError[w_Index](
		b_ErrorTrig			:= NOT(get.b_Type12_OK),
		out_ST_Error			:= a_ActiveEvents[w_Index],
		w_ErrorID					:= 1,
		e_ObjectID				:= eObject_ID.SurgeProtection,
		s_Message				:= 'Type 1+2 Fault',
		e_sev					:= eseverity.warning,
		e_ErrAckAccess		:= eErrAckAccess.VDL
	);
	w_Index := w_Index +1;
	
(*Type3 warning*)			AddError[w_Index](
		b_ErrorTrig			:= NOT(get.b_Type3_OK),
		out_ST_Error			:= a_ActiveEvents[w_Index],
		w_ErrorID					:= 2,
		s_Message				:= 'Type 3 Fault',
		e_sev					:= eseverity.warning,
		e_ErrAckAccess		:= eErrAckAccess.VDL
	);
	w_Index := w_Index +1;
END_METHOD

END_FUNCTION_BLOCK

// ---- POUs/Objects/ProtectionSystems/ResidualCurrentMonitoring/FB_RCMonitor.TcPOU
FUNCTION_BLOCK FB_RCMonitor
VAR_OUTPUT
	get				: ST_ResidualCurrentMonitor_get;
END_VAR

VAR CONSTANT
	w_ID			: WORD := eObject_ID.RCM;
END_VAR

VAR
	b_prewarningOK	AT %I* : BOOL;
	b_PowerOff		AT %Q* : BOOL;
END_VAR

get.b_prewarning := NOT(b_prewarningOK);

METHOD GetDiagnostics
VAR_IN_OUT
	AddError		: ARRAY [*] OF FB_AddErrorST;
	a_ActiveEvents	: ARRAY [*] OF ST_ErrorStruct;
	w_Index			: WORD;
END_VAR
(*OBSOLETE prewarning*)			AddError[w_Index](
		b_ErrorTrig			:= FALSE,//get.b_prewarning,
		out_ST_Error			:= a_ActiveEvents[w_Index],
		w_ErrorID					:= 1,
		e_ObjectID				:= eobject_ID.RCM,
		s_Message				:= 'RCD prewarning',
		e_sev					:= eseverity.warning,
		e_ErrAckAccess		:= eErrAckAccess.General,
		b_AutoClear 			:= TRUE,
	);
	w_Index := w_Index +1;
END_METHOD

METHOD Reset : BOOL
VAR_INPUT
END_VAR

VAR_INST
	ton_ResetPower		: Ton := (PT := T#500MS);
	b_toggle			: BOOL;
END_VAR
Reset := FALSE;
ton_ResetPower(IN:= NOT ton_ResetPower.Q);

IF ton_ResetPower.Q THEN
	b_toggle := NOT b_toggle;
END_IF

IF get.b_prewarning THEN
	b_PowerOff := b_toggle;
ELSE
	b_PowerOff := FALSE;
	Reset :=  TRUE;
END_IF
END_METHOD

END_FUNCTION_BLOCK

// ---- POUs/Objects/ProtectionSystems/OvercurrentProtection/FB_OvercurrentProtection.TcPOU
FUNCTION_BLOCK FB_OvercurrentProtection
VAR_IN_OUT CONSTANT
	st_params 			: ST_overcurrentprotection_Params;
	powermonitor		: ST_Powermonitor_get;
END_VAR

VAR_OUTPUT
	get					: ST_Overcurrentprotection_get;
END_VAR

VAR_INPUT
	set							: ST_Overcurrentprotection_set;
	b_enable					: BOOL := TRUE;
	b_InputSectionAvailable 	: BOOL;
	b_thirdOutputAvailable 		: BOOL;
END_VAR

VAR
	b_reset 					: BOOL;
	//OvercurrentTest				: FB_Overcurrentdetect;
	//r_test		: REAL;
END_VAR

IF b_enable THEN
	CheckOvercurrent(get, set, b_reset);
END_IF

IF b_InputSectionAvailable THEN
	get.r_TotalInputCurrentLimit := set.ui_PowerlockInputCurrentLimit[1] + set.ui_PowerlockInputCurrentLimit[2];
END_IF

get.r_TotalOutputCurrentLimit := 
	set.ui_PowerlockOutputCurrentLimit[1] + 
	set.ui_PowerlockOutputCurrentLimit[2] + 
	set.ui_PowerlockOutputCurrentLimit[3] * TO_BYTE(b_thirdOutputAvailable);

METHOD CheckOvercurrent : BOOL

VAR_IN_OUT
	get			: ST_OvercurrentProtection_get;
END_VAR

VAR_IN_OUT CONSTANT
	set 		: ST_OvercurrentProtection_set;
	reset		: BOOL;
END_VAR

VAR
	i : BYTE;
	j : BYTE;
	phase		: Phases;
END_VAR

VAR_INST
	r_lastcurrent		: REAL;
	sr_outputAlarm		: SR;
	sr_inputAlarm		: SR;
END_VAR
get.b_InputWarning := FALSE;
get.b_OutputWarning := FALSE;
get.b_InputAlarm := FALSE;
get.b_OutputAlarm := FALSE;

//Inputs
FOR j:=1 TO 2 DO //loop through powerlock sets
	FOR phase:=1 TO 4 DO //loop through powerlocks
		get.events.Input[j][phase](b_reset := reset,
				r_In := ABS(powermonitor.InputField.Powerlock[j].ar_Current[phase]),
				ui_Ik := st_params.ui_Ik,
				ui_gain := st_params.ui_gain,
				ui_RatedCurrent := LIMIT(0, TO_UINT(set.ui_PowerlockInputCurrentLimit[j]), st_params.ui_Irated),
				t_MaxPickupTime := TO_TIME(TO_REAL(st_params.ui_OCPtripTime)*1000),
				);

		IF get.Events.Input[j][phase].r_MaxCurrentDetected > r_lastcurrent THEN
			r_lastcurrent := get.Events.input[j][phase].r_MaxCurrentDetected;
			get.r_PeakCurrent := r_lastcurrent;
			get.t_PeakCurrentDuration := get.Events.input[j][phase].t_MaxTimeActive;
			get.s_locationPeak := CONCAT(CONCAT(CONCAT('Input group: ', TO_STRING(j)),' '), TO_STRING(phase));
		END_IF	
		IF get.events.input[j][phase].b_warning THEN
			get.b_inputwarning := TRUE;
		END_IF
		IF get.events.Input[j][phase].b_alarm THEN
			get.b_InputAlarm := TRUE;
		END_IF
	END_FOR
END_FOR

//Outputs
FOR j:=1 TO 3 DO
	FOR phase:=1 TO 4 DO 
		get.events.Output[j][phase](b_reset := reset,
			r_In := ABS(powermonitor.OutputField.Powerlock[j].ar_Current[phase]),
			ui_Ik := st_params.ui_Ik,
			ui_gain := st_params.ui_gain,
			ui_RatedCurrent := LIMIT(0, TO_UINT(set.ui_PowerlockOutputCurrentLimit[j]), st_params.ui_Irated),
			t_MaxPickupTime := TO_TIME(TO_REAL(st_params.ui_OCPtripTime)*1000)
			);
		IF get.Events.output[j][phase].r_MaxCurrentDetected > r_lastcurrent THEN
			r_lastcurrent := get.Events.output[j][phase].r_MaxCurrentDetected;
			get.r_PeakCurrent := r_lastcurrent;
			get.t_PeakCurrentDuration := get.Events.output[j][phase].t_MaxTimeActive;
			get.s_locationPeak := CONCAT(CONCAT(CONCAT('Output group: ', TO_STRING(j)),' '), TO_STRING(phase));
		END_IF
			
		IF get.events.Output[j][phase].b_warning THEN
			get.b_outputwarning := TRUE;
		END_IF
		IF get.events.Output[j][phase].b_alarm THEN
			get.b_OutputAlarm := TRUE;
		END_IF
	END_FOR
END_FOR
END_METHOD

METHOD PUBLIC GetDiagnostics
VAR_IN_OUT
	AddError		: ARRAY [*] OF FB_AddErrorST;
	a_ActiveEvents	: ARRAY [*] OF ST_ErrorStruct;
	w_Index			: WORD;
END_VAR

VAR	
		
	i : UINT; 
END_VAR

VAR_INST
	index : WORD;
END_VAR
(*OVC PROTECTION*)
//INPUTS
index := w_index;
FOR i:= 1 TO 2 DO
	//Warnings
	(*Input set1 L1*) 	AddError[w_Index](
			b_ErrorTrig			:= Get.Events.Input[i][phases.L1].b_warning,
			out_ST_Error			:= a_ActiveEvents[w_Index],
			w_ErrorID					:= ((i -1) * 8) + 1,
			e_ObjectID				:= eObject_ID.OCP,
			s_Message				:= ConcatMultiString(s1:= 'warning: input ',
										s2:= TO_STRING(i),
			 							s3:= ' - L1: ',
										s4:= TO_STRING(Get.Events.Input[i][phases.L1].ui_actLoad),
										s5:= ' %, remaining time ',
										s6:= TO_STRING(Get.Events.Input[i][phases.L1].t_RemainingTime)),
			e_sev					:= eseverity.Warning,
			e_ErrAckAccess		:= eErrAckAccess.operator,
			b_autoClear			:= TRUE
			);
		w_Index := w_Index +1;
	(*Input set1 L2*) 	AddError[w_Index](
			b_ErrorTrig			:= Get.Events.Input[i][phases.L2].b_warning,
			out_ST_Error			:= a_ActiveEvents[w_Index],
			w_ErrorID					:= ((i -1) * 8) + 2,
			s_Message				:= ConcatMultiString(s1:= 'warning: input ',
										s2:= TO_STRING(i),
			 							s3:= ' - L2: ',
										s4:= TO_STRING(Get.Events.Input[i][phases.L2].ui_actLoad),
										s5:= ' %, remaining time ',
										s6:= TO_STRING(Get.Events.Input[i][phases.L2].t_RemainingTime)),
			e_sev					:= eseverity.Warning,
			e_ErrAckAccess		:= eErrAckAccess.operator,
			b_autoClear			:= TRUE
			);
		w_Index := w_Index +1;
	(*Input set1 L3*) 	AddError[w_Index](
			b_ErrorTrig			:= Get.Events.Input[i][phases.L3].b_warning,
			out_ST_Error			:= a_ActiveEvents[w_Index],
			w_ErrorID					:= ((i -1) * 8) + 3,
			s_Message				:= ConcatMultiString(s1:= 'warning: input ',
										s2:= TO_STRING(i),
			 							s3:= ' - L3: ',
										s4:= TO_STRING(Get.Events.Input[i][phases.L3].ui_actLoad),
										s5:= ' %, remaining time ',
										s6:= TO_STRING(Get.Events.Input[i][phases.L3].t_RemainingTime)),
			e_sev					:= eseverity.Warning,
			e_ErrAckAccess		:= eErrAckAccess.operator,
			b_autoClear			:= TRUE
			);
		w_Index := w_Index +1;
	(*Input set1 N*) 	AddError[w_Index](
			b_ErrorTrig			:= Get.Events.Input[i][phases.N].b_warning,
			out_ST_Error			:= a_ActiveEvents[w_Index],
			w_ErrorID					:= ((i -1) * 8) + 4,
			s_Message				:= ConcatMultiString(s1:= 'warning: input ',
										s2:= TO_STRING(i),
			 							s3:= ' - Neutral: ',
										s4:= TO_STRING(Get.Events.Input[i][phases.N].ui_actLoad),
										s5:= ' %, remaining time ',
										s6:= TO_STRING(Get.Events.Input[i][phases.N].t_RemainingTime)),
			e_sev					:= eseverity.Warning,
			e_ErrAckAccess		:= eErrAckAccess.operator,
			b_autoClear			:= TRUE
			);
		w_Index := w_Index +1;
		
		//ALARMS
	(*Input set1 L1*) 	AddError[w_Index](
			b_ErrorTrig			:= Get.Events.Input[i][phases.L1].b_alarm,
			out_ST_Error			:= a_ActiveEvents[w_Index],
			w_ErrorID					:= ((i -1) * 8) + 5,
			s_Message				:= ConcatMultiString(s1:= 'alarm: input ',
										s2:= TO_STRING(i),
			 							s3:= ' - L1: ',
										s4:= LREAL_TO_FMTSTR(Get.Events.Input[i][phases.L1].r_MaxCurrentDetected,1, TRUE),
										s5:= ' A for ',
										s6:= TO_STRING(Get.Events.Input[i][phases.L1].t_MaxTimeActive)),
			e_sev					:= eseverity.Warning,
			e_ErrAckAccess		:= eErrAckAccess.operator
			);
		w_Index := w_Index +1;
	(*Input set1 L2*) 	AddError[w_Index](
			b_ErrorTrig			:= Get.Events.Input[i][phases.L2].b_alarm,
			out_ST_Error			:= a_ActiveEvents[w_Index],
			w_ErrorID					:= ((i -1) * 8) + 6,
			s_Message				:= ConcatMultiString(s1:= 'alarm: input ',
										s2:= TO_STRING(i),
			 							s3:= ' - L2: ',
										s4:= LREAL_TO_FMTSTR(Get.Events.Input[i][phases.L2].r_MaxCurrentDetected,1, TRUE),
										s5:= ' A for ',
										s6:= TO_STRING(Get.Events.Input[i][phases.L2].t_MaxTimeActive)),
			e_sev					:= eseverity.Warning,
			e_ErrAckAccess		:= eErrAckAccess.operator
			);
		w_Index := w_Index +1;
	(*Input set1 L3*) 	AddError[w_Index](
			b_ErrorTrig			:= Get.Events.Input[i][phases.L3].b_alarm,
			out_ST_Error			:= a_ActiveEvents[w_Index],
			w_ErrorID					:= ((i -1) * 8) + 7,
			s_Message				:= ConcatMultiString(s1:= 'alarm: input ',
										s2:= TO_STRING(i),
			 							s3:= ' - L3: ',
										s4:= LREAL_TO_FMTSTR(Get.Events.Input[i][phases.L3].r_MaxCurrentDetected,1, TRUE),
										s5:= ' A for ',
										s6:= TO_STRING(Get.Events.Input[i][phases.L3].t_MaxTimeActive)),
			e_sev					:= eseverity.Warning,
			e_ErrAckAccess		:= eErrAckAccess.operator
			);
		w_Index := w_Index +1;
	(*Input set1 N*) 	AddError[w_Index](
			b_ErrorTrig			:= Get.Events.Input[i][phases.N].b_alarm,
			out_ST_Error			:= a_ActiveEvents[w_Index],
			w_ErrorID					:= ((i -1) * 8) + 8,
			s_Message				:= ConcatMultiString(s1:= 'alarm: input ',
										s2:= TO_STRING(i),
			 							s3:= ' - N: ',
										s4:= LREAL_TO_FMTSTR(Get.Events.Input[i][phases.N].r_MaxCurrentDetected,1, TRUE),
										s5:= ' A for ',
										s6:= TO_STRING(Get.Events.Input[i][phases.N].t_MaxTimeActive)),
			e_sev					:= eseverity.Warning,
			e_ErrAckAccess		:= eErrAckAccess.operator
			);
		w_Index := w_Index +1;
END_FOR

//OUTPUTS
FOR i:= 1 TO 3 DO
	//Warnings
	(*Input set1 L1*) 	AddError[w_Index](
			b_ErrorTrig			:= Get.Events.Output[i][phases.L1].b_warning,
			out_ST_Error			:= a_ActiveEvents[w_Index],
			w_ErrorID					:= ((i -1) * 8) + 17,
			s_Message				:= ConcatMultiString(s1:= 'warning: output ',
										s2:= TO_STRING(i),
			 							s3:= ' - L1: ',
										s4:= TO_STRING(Get.Events.Output[i][phases.L1].ui_actLoad),
										s5:= ' %, remaining time ',
										s6:= TO_STRING(Get.Events.Output[i][phases.L1].t_RemainingTime)),
			e_sev					:= eseverity.Warning,
			e_ErrAckAccess		:= eErrAckAccess.operator,
			b_autoClear			:= TRUE
			);
		w_Index := w_Index +1;
	(*Input set1 L2*) 	AddError[w_Index](
			b_ErrorTrig			:= Get.Events.Output[i][phases.L2].b_warning,
			out_ST_Error			:= a_ActiveEvents[w_Index],
			w_ErrorID					:= ((i -1) * 8) + 18,
			s_Message				:= ConcatMultiString(s1:= 'warning: output ',
										s2:= TO_STRING(i),
			 							s3:= ' - L2: ',
										s4:= TO_STRING(Get.Events.Output[i][phases.L2].ui_actLoad),
										s5:= ' %, remaining time ',
										s6:= TO_STRING(Get.Events.Output[i][phases.L2].t_RemainingTime)),
			e_sev					:= eseverity.Warning,
			e_ErrAckAccess		:= eErrAckAccess.operator,
			b_autoClear			:= TRUE
			);
		w_Index := w_Index +1;
	(*Input set1 L3*) 	AddError[w_Index](
			b_ErrorTrig			:= Get.Events.Output[i][phases.L3].b_warning,
			out_ST_Error			:= a_ActiveEvents[w_Index],
			w_ErrorID					:= ((i -1) * 8) + 19,
			s_Message				:= ConcatMultiString(s1:= 'warning: output ',
										s2:= TO_STRING(i),
			 							s3:= ' - L3: ',
										s4:= TO_STRING(Get.Events.Output[i][phases.L3].ui_actLoad),
										s5:= ' %, remaining time ',
										s6:= TO_STRING(Get.Events.Output[i][phases.L3].t_RemainingTime)),
			e_sev					:= eseverity.Warning,
			e_ErrAckAccess		:= eErrAckAccess.operator,
			b_autoClear			:= TRUE
			);
		w_Index := w_Index +1;
	(*Input set1 N*) 	AddError[w_Index](
			b_ErrorTrig			:= Get.Events.Output[i][phases.N].b_warning,
			out_ST_Error			:= a_ActiveEvents[w_Index],
			w_ErrorID				:= ((i -1) * 8) + 20,
			s_Message				:= ConcatMultiString(s1:= 'warning: output ',
										s2:= TO_STRING(i),
			 							s3:= ' - N: ',
										s4:= TO_STRING(Get.Events.Output[i][phases.N].ui_actLoad),
										s5:= ' %, remaining time ',
										s6:= TO_STRING(Get.Events.Output[i][phases.N].t_RemainingTime)),
			e_sev					:= eseverity.Warning,
			e_ErrAckAccess		:= eErrAckAccess.operator,
			b_autoClear			:= TRUE
			);
		w_Index := w_Index +1;
		
		//ALARMS					
	(*Output set1 L1*) 	AddError[w_Index](
			b_ErrorTrig			:= Get.Events.Output[i][phases.L1].b_alarm,
			out_ST_Error			:= a_ActiveEvents[w_Index],
			w_ErrorID					:= ((i -1) * 8) + 21,
			s_Message				:= ConcatMultiString(s1:= 'alarm: output ',
										s2:= TO_STRING(i),
			 							s3:= ' - L1: ',
										s4:= LREAL_TO_FMTSTR(Get.Events.output[i][phases.L1].r_MaxCurrentDetected,1, TRUE),
										s5:= ' A for ',
										s6:= TO_STRING(Get.Events.Output[i][phases.L1].t_MaxTimeActive)),
			e_sev					:= eseverity.Normalshutdown,
			t_triggerTime			:= st_params.OutputNormalShutdownDelay,
			e_ErrAckAccess		:= eErrAckAccess.operator
			);
		w_Index := w_Index +1;
	(*Output set1 L2*) 	AddError[w_Index](
			b_ErrorTrig			:= Get.Events.Output[i][phases.L2].b_alarm,
			out_ST_Error			:= a_ActiveEvents[w_Index],
			w_ErrorID					:= ((i -1) * 8) + 22,
			s_Message				:= ConcatMultiString(s1:= 'alarm: output ',
										s2:= TO_STRING(i),
			 							s3:= ' - L2: ',
										s4:= LREAL_TO_FMTSTR(Get.Events.output[i][phases.L2].r_MaxCurrentDetected,1, TRUE),
										s5:= ' A for ',
										s6:= TO_STRING(Get.Events.Output[i][phases.L2].t_MaxTimeActive)),
			e_sev					:= eseverity.Normalshutdown,
			t_triggerTime			:= st_params.OutputNormalShutdownDelay,
			);
		w_Index := w_Index +1;
	(*Output set1 L3*) 	AddError[w_Index](
			b_ErrorTrig			:= Get.Events.Output[i][phases.L3].b_alarm,
			out_ST_Error			:= a_ActiveEvents[w_Index],
			w_ErrorID					:= ((i -1) * 8) + 23,
			s_Message				:= ConcatMultiString(s1:= 'alarm: output ',
										s2:= TO_STRING(i),
			 							s3:= ' - L3: ',
										s4:= LREAL_TO_FMTSTR(Get.Events.output[i][phases.L3].r_MaxCurrentDetected,1, TRUE),
										s5:= ' A for ',
										s6:= TO_STRING(Get.Events.Output[i][phases.L3].t_MaxTimeActive)),
			e_sev					:= eseverity.Normalshutdown,
			t_triggerTime			:= st_params.OutputNormalShutdownDelay,
			e_ErrAckAccess		:= eErrAckAccess.operator
			);
		w_Index := w_Index +1;
	(*Output set1 N*) 	AddError[w_Index](
			b_ErrorTrig			:= Get.Events.output[i][phases.N].b_alarm,
			out_ST_Error			:= a_ActiveEvents[w_Index],
			w_ErrorID					:= ((i -1) * 8) + 24,
			s_Message				:= ConcatMultiString(s1:= 'alarm: output ',
										s2:= TO_STRING(i),
			 							s3:= ' - N: ',
										s4:= LREAL_TO_FMTSTR(Get.Events.output[i][phases.N].r_MaxCurrentDetected,1, TRUE),
										s5:= ' A for ',
										s6:= TO_STRING(Get.Events.Output[i][phases.N].t_MaxTimeActive)),
			e_sev					:= eseverity.Normalshutdown,
			t_triggerTime 			:= st_params.OutputNormalShutdownDelay,
			e_ErrAckAccess		:= eErrAckAccess.operator
			);
		w_Index := w_Index +1;
END_FOR	

(*output MCCB triggered*) 	AddError[w_Index](
			b_ErrorTrig				:= Get.b_OutputAlarm,
			out_ST_Error			:= a_ActiveEvents[w_Index],
			w_ErrorID				:= 41,
			s_Message				:= ConcatMultiString(s1:= 'Output MCCB trip. Phase: ',
										s2:= get.s_locationPeak,
			 							s3:= ', peakcurrent: ',
										s4:= LREAL_TO_FMTSTR(get.r_PeakCurrent,1, TRUE),
										s5:= ' A for ',
										s6:= TO_STRING(get.t_PeakCurrentDuration)),
			e_sev					:= eseverity.Warning
			);
		w_Index := w_Index +1;
END_METHOD

METHOD Reset : BOOL
VAR_INPUT
END_VAR

VAR_INST
	counter : INT;
END_VAR
reset := FALSE;


//reset values if it was triggered by an alarm
IF get.b_InputAlarm OR get.b_OutputAlarm OR get.r_PeakCurrent <>0 THEN
	get.r_PeakCurrent := 0;
	get.t_PeakCurrentDuration := T#0S;
	get.s_locationPeak := '';
	b_reset := TRUE;
	counter := counter +1;
ELSE
	b_reset := FALSE;
	reset := NOT b_reset;
END_IF
END_METHOD

END_FUNCTION_BLOCK

// ---- POUs/Functions-FBs-Programs/_generalFunctions/ConcatMultiString.TcPOU
FUNCTION ConcatMultiString : STRING
VAR_INPUT
	s1: STRING;
	s2: STRING;
	s3: STRING;
	s4: STRING;
	s5: STRING;
	s6: STRING;
END_VAR
VAR
END_VAR

ConcatMultiString := CONCAT(s1, CONCAT(s2, CONCAT(s3, CONCAT(s4, CONCAT(s5, s6)))));

END_FUNCTION

// ---- POUs/Objects/Enclosure/FB_Enclosure.TcPOU
FUNCTION_BLOCK FB_Enclosure
VAR_IN_OUT CONSTANT
	st_params		: ST_Enclosure_params;
END_VAR

VAR_OUTPUT
	get					: ST_Enclosure_Get;
END_VAR

VAR_INPUT
	ledstrip			: FB_ledstrip;
	set					: ST_Enclosure_set;
END_VAR

VAR
	
	climate						: FB_enclosureClimate;
	doors						: FB_DoorsNlocks;
END_VAR

ledstrip(st_params := st_params.ledstrip, get => get.ledstrip, brightness := set.by_LedBrightness);

climate( get => get.climate, st_params:= st_params.Climate);

doors(get => get.doors);

METHOD PUBLIC GetDiagnostics
VAR_IN_OUT
	AddError		: ARRAY [*] OF FB_AddErrorST;
	a_ActiveEvents	: ARRAY [*] OF ST_ErrorStruct;
	w_Index			: WORD;
END_VAR

VAR_OUTPUT
	b_errorActive	: BOOL;
	b_warningActive	: BOOL;
END_VAR

VAR
	by_errCt	: BYTE;
	by_warnCt	: BYTE;
END_VAR
Climate.GetDiagnostics(Adderror := AddError, a_ActiveEvents := a_ActiveEvents, w_Index := w_index);
Doors.GetDiagnostics(Adderror := AddError, a_ActiveEvents := a_ActiveEvents, w_Index := w_index);
Ledstrip.GetDiagnostics(Adderror := AddError, a_ActiveEvents := a_ActiveEvents, w_Index := w_index);
END_METHOD

METHOD GetWearCounters : BOOL
VAR_INST
	ControlCabinetDoorSwitch	:	FB_Varlogger;
	ClientPanelDoorSwitch		:	FB_Varlogger;
	
END_VAR
ControlCabinetDoorSwitch(	TriggerInput := NOT get.doors.b_ControlPanelDoorClosed, 
							LogItemGroup :=  eLogItemGroupID.Enclosure, 
							LogItemName := 'CtrlCabDoorSwCnt', 
							LogType := elogtypes.TrackCycles);		
												
ClientPanelDoorSwitch(	TriggerInput := NOT get.doors.b_ClientpanelDoorClosed, 
						LogItemGroup :=  eLogItemGroupID.Enclosure, 
						LogItemName := 'ClientPnlDoorSwCnt', 
						LogType := eLogtypes.TrackCycles);
END_METHOD

END_FUNCTION_BLOCK

// ---- POUs/Objects/Enclosure/LedIndicator/FB_Ledstrip.TcPOU
FUNCTION_BLOCK FB_Ledstrip
VAR_INPUT
	brightness						: BYTE; // in 
END_VAR

VAR_IN_OUT CONSTANT
	st_params				: st_ledstrip_params;
END_VAR

VAR_OUTPUT
	get 					: st_ledstrip_get;
END_VAR
VAR
	ledArduino				: FB_LedArduino;
	ledBeckhoff				: FB_ledBeckhoff;
	MachineData				: ST_Ledstrip_MachineData;
END_VAR

ledbeckhoff(Machinedata := Machinedata, st_params := st_params, Brightness := brightness, DemoMode := GVL.b_LEDDemoMode);
ledArduino(enable := NOT ledbeckhoff.Ready, MachineData := Machinedata, st_params := st_params, brightness := brightness);

IF ledbeckhoff.Ready THEN
	get := ledbeckhoff.get;
ELSE
	get := ledArduino.get;
END_IF

METHOD PUBLIC GetDiagnostics
VAR_IN_OUT
	AddError		: ARRAY [*] OF FB_AddErrorST;
	a_ActiveEvents	: ARRAY [*] OF ST_ErrorStruct;
	w_Index			: WORD;
END_VAR

VAR_OUTPUT
	b_errorActive	: BOOL;
	b_warningActive	: BOOL;
END_VAR

VAR
	by_errCt	: BYTE;
	by_warnCt	: BYTE;
END_VAR
	(*LED Error*)		AddError[w_Index](
		b_ErrorTrig			:= get.b_error,
		out_ST_Error			:= a_ActiveEvents[w_Index],
		w_ErrorID					:= 1,
		e_ObjectID				:=  eObject_ID.Enclosure_LED,
		s_Message				:= 'LED error',
		e_sev					:= eseverity.info,
		b_AutoClear			:= TRUE
		);
		w_Index := w_Index +1;
END_METHOD

METHOD SetMachineStatus : BOOL
VAR_INPUT
	b_Error 		: BOOL;
	b_Warning		: BOOL;
	b_Attention		: BOOL;
	b_Normal		: BOOL;
	b_Off			: BOOL;
	r_Soc			: REAL;
	r_DCcurrent		: REAL;
END_VAR

VAR_INST
	r_socDemo	: REAL := 30;
	r_CurrentDemo : REAL := 0;
END_VAR
IF b_off THEN
	machinedata.e_systemStatus := eSystemStatus.off;
ELSIF b_Error THEN
	machinedata.e_systemStatus := eSystemStatus.error;
ELSIF b_warning THEN
	machinedata.e_systemStatus := eSystemStatus.warning;
ELSIF b_attention THEN
	machinedata.e_systemStatus := eSystemStatus.attention;
ELSIF b_normal THEN
	machinedata.e_systemStatus := eSystemStatus.normal;
ELSE
	machinedata.e_systemStatus := eSystemStatus.neutral;
END_IF

MachineData.r_SOC := r_soc;
MachineData.r_DCCurrent := r_DCcurrent;
END_METHOD

END_FUNCTION_BLOCK

// ---- POUs/Objects/Enclosure/LedIndicator/ArduinoController/FB_LedArduino.TcPOU
FUNCTION_BLOCK FB_LedArduino
VAR_INPUT
	brightness					: BYTE; // in %
	enable					: BOOL := TRUE;
END_VAR

VAR_IN_OUT CONSTANT
	MachineData						: ST_Ledstrip_MachineData;
	st_params						: st_ledstrip_params;
END_VAR

VAR CONSTANT
	w_ID						: WORD := eObject_ID.Enclosure_LED;
END_VAR

VAR_OUTPUT
	get						: ST_Ledstrip_get;
END_VAR

VAR
	Write						: TON;
	w_NoRegisters				: WORD;
	CommFaultOffDelay			: TOF;
	aw_LED_ModbusOutputRegs		: ARRAY [0..10] OF WORD;
	WriteRegs					: FB_MBWriteRegs;
	t_RefreshTime				: TIME := T#1S;
	t_TimeOut					: TIME := T#1S;
END_VAR

SetData();

IF st_params.ColorOrder = eColororder.GRB THEN
	w_NoRegisters		:= 7;
ELSE
	w_NoRegisters		:= 6;
END_IF

IF enable THEN
	Write(IN:= NOT write.Q, PT := t_RefreshTime);
	CommFaultOffDelay(IN:= writeregs.bError, PT := T#5S, Q => get.b_error);
	
	WriteRegs(sIPAddr := st_params.IP,
		nTCPPort := 502,
		nUnitID := 16#FF,
		nQuantity := w_NoRegisters,
		nMBaddr := 0,
		cbLength := SIZEOF(aw_LED_ModbusOutputRegs),
		pSrcAddr := ADR(aw_LED_ModbusOutputRegs),
		bExecute := Write.Q,
		tTimeOut := t_Timeout);	
END_IF

METHOD PUBLIC GetDiagnostics
VAR_IN_OUT
	AddError		: ARRAY [*] OF FB_AddErrorST;
	a_ActiveEvents	: ARRAY [*] OF ST_ErrorStruct;
	w_Index			: WORD;
END_VAR

VAR_OUTPUT
	b_errorActive	: BOOL;
	b_warningActive	: BOOL;
END_VAR

VAR
	by_errCt	: BYTE;
	by_warnCt	: BYTE;
END_VAR
	(*Led Com fault*)		AddError[w_Index](
		b_ErrorTrig			:= get.b_error,
		out_ST_Error			:= a_ActiveEvents[w_Index],
		w_ErrorID					:= 1,
		e_ObjectID				:=  eObject_ID.Enclosure_LED,
		s_Message				:= 'communication fault',
		e_sev					:= eseverity.info,
		b_AutoClear			:= TRUE
		);
		w_Index := w_Index +1;
END_METHOD

METHOD PUBLIC Reset : BOOL

VAR_INST
	ton_ResetPulse			: TON := (pt:=T#500MS);

END_VAR
IF get.b_error THEN
	ton_resetPulse(IN:= NOT ton_ResetPulse.Q);
	enable := ton_ResetPulse.Q;
ELSE
	enable := TRUE;
END_IF

reset := NOT get.b_error;
END_METHOD

METHOD PRIVATE SetData


VAR
	by_Status 					: BYTE;
	by_mode						: BYTE := 0;
END_VAR

VAR_INST
	TON_ledstripColorPulse			: TON := (PT:=T#500MS);
	b_toggle						: BOOL;
END_VAR
TON_ledstripColorPulse(IN:= NOT TON_ledstripColorPulse.Q);
IF ton_ledstripColorPulse.Q THEN
	b_toggle := NOT b_toggle;
END_IF


 // Get status
CASE machinedata.e_systemStatus OF
	eSystemstatus.error: by_Status := 4;
	eSystemstatus.warning: by_Status := 3;
	eSystemstatus.attention: by_Status := 2;
	eSystemstatus.normal: by_Status := 1;
	eSystemstatus.neutral: by_Status := 0;
END_CASE

IF machinedata.r_DCCurrent < -10 THEN
	by_mode := 1; //charging
ELSIF machinedata.r_DCCurrent > 10 THEN
	by_mode := 2; //discharging
ELSE
	by_mode := 0; // idle
END_IF


// Fill in regs
aw_LED_ModbusOutputRegs[0] := TO_WORD(MAX(LIMIT(0,machinedata.r_SOC,100) *2.55,1));   				// Battery usable state of charge (0.1%)
aw_LED_ModbusOutputRegs[1] := TO_WORD(by_Status); // Battery status (0: Neutral, 1: Normal, 2: attention, 3: Warning, 4: Error)
aw_LED_ModbusOutputRegs[2] := TO_WORD(by_mode);	// 0 = idle, 1 = charging, 2 = discharging				
aw_LED_ModbusOutputRegs[3] := TO_WORD(SEL(machinedata.e_systemStatus = 0, LIMIT(10, brightness, 100), 0) * 2.55); 					// LED strip brightness (0-255)
aw_LED_ModbusOutputRegs[4] := st_params.Numleds; 	
aw_LED_ModbusOutputRegs[5] := 0; 	  
aw_LED_ModbusOutputRegs[6] := st_params.ColorOrder;
END_METHOD

END_FUNCTION_BLOCK

// ---- POUs/Objects/Enclosure/LedIndicator/BeckhoffController/FB_LedBeckhoff.TcPOU
FUNCTION_BLOCK FB_LedBeckhoff
VAR_INPUT
	Brightness				: BYTE;
	DemoMode				: BOOL;
END_VAR
VAR_OUTPUT
	get 					: st_ledstrip_get;
	Ready					: BOOL;			
END_VAR

VAR_IN_OUT CONSTANT
	MachineData				: ST_Ledstrip_machineData;
	st_params				: st_ledstrip_params;
END_VAR

VAR	
	EL2574State		AT %I* 	: UINT;
	st_LEDStatus	AT %I* 	: LEDStatus;
	st_LEDControl	AT %Q* 	: LEDControl;	
	ton_LEDdataSend		: ton := (PT:=T#300MS);
	LedsToAnimate		: BYTE		:= 5;

	ui_ActiveLeds		: UINT;
	e_LEDSteps			: eLEDSteps;
	ui_oldSOC			: UINT;
	ui_SOC 				: UINT;
	SFCStep				: UINT;
	LedBusy				: TOF := (PT := T#50MS);
	AnimationReady		: BOOL;
	
	bufferReady			: BOOL;
	ReadyToTransmit		: BOOL;
	
	GradientToggle		: BOOL;
	DemoSoc				: UINT := 50;
	DemoSocPulse		: TON := (PT:= T#500MS);
	DemoCharging		: BOOL;
END_VAR

ready := EL2574State.3;
LedBusy(IN := st_ledStatus.busy OR st_ledstatus.transmit OR st_ledstatus.error OR st_LEDControl.Execute);



IF ready THEN //AND ton_CycleTime.Q THEN
	get.BeckhoffLed := TRUE;
	
	//get system state error
	IF Machinedata.e_systemStatus = eSystemStatus.error THEN
		ui_SOC := 100;
	ELSE
		ui_SOC := REAL_TO_UINT (Machinedata.r_soc);
	END_IF
	
	//set ledstrip error to system
	get.b_Error := st_LEDStatus.error;
	
	//SOc and corresponding leds
	
	ui_ActiveLeds:= ((st_params.Numleds * ui_SOC)/100);
	
//	IF MachineData.e_systemStatus = 0 THEN
//		e_LEDSteps := eLEDSteps.initialise;
//	END_IF
	
	//setup color values and no of led according to soc. 
	CASE e_LEDSteps OF	
		eLEDSteps.initialise:
			st_LEDControl.command := 2; //Clear
			st_LEDControl.length := st_params.Numleds;
			st_LEDControl.index := 0;

			IF NOT ledbusy.Q THEN
				st_LEDControl.execute := NOT st_LEDControl.execute;
				st_LEDControl.update  := NOT st_LEDControl.update;
				e_LEDSteps := eLEDSteps.running;	
			END_IF
						

		eLEDSteps.running:	
			st_LEDControl.UPDATE 	:= FALSE;
			st_LEDControl.Execute 	:= FALSE;
			CASE SFCStep OF 
				0: 	BufferReady := FALSE;
					ReadyToTransmit := FALSE;
					st_LEDControl.command	:= 2; //Clear
					
					IF NOT LedBusy.Q THEN
						st_LEDControl.Execute 	:= NOT st_LEDControl.Execute;
						SFCStep := SEL(DemoMode, 1,2);
					END_IF
						
				1:	st_LEDControl.command	:= 1; //fill
					st_LEDControl.length 	:= ui_ActiveLeds;
					st_LEDControl.index		:= 0;
					st_LEDcontrol.parameter := 0;
					st_LEDControl.color 	:= setcolor(brightness);
					
					IF NOT LedBusy.Q THEN
						st_LEDControl.Execute 	:= NOT st_LEDControl.Execute;
						SFCStep := 3;
					END_IF
				2: //demo mode
					DemoSocPulse(IN := NOT DemoSocPulse.Q);
					IF DemoSocPulse.Q THEN
						IF DemoSoc <= 50 THEN
							DemoCharging := TRUE;
						ELSIF DemoSoc >= st_Params.Numleds THEN
							DemoCharging := FALSE;
						END_IF
						
						DemoSoc := DemoSoc + SEL(democharging, -1, 1);
					END_IF
					
					IF NOT DemoMode THEN SfcSTEP := 0; END_IF;
					st_LEDControl.length 	:= demosoc;
					st_LEDControl.index		:= 0;
					st_LEDControl.color.blue:= 0;
					
					IF NOT GradientToggle THEN
						st_LEDControl.command	:= 8; //fill
						st_LEDControl.color.Green:= 0;
						st_LEDControl.color.red:= brightness;
					ELSE
						st_LEDControl.command	:= 9; //fill
						st_LEDControl.color.Green:= brightness;
						st_LEDControl.color.red:= 0;
					END_IF
					
					IF NOT LedBusy.Q THEN
						st_LEDControl.Execute 	:= NOT st_LEDControl.Execute;
						
